  MoveL 3100 to (-5.96, 26.09, 135) mm, rotated rx -180 ry 0 rz 180 deg; joints [-155.969, -46.941, -94.947, 29.54, 55.687, -17.716]
  Call Extruder(28979.31277)
  MoveL 3101 to (-11.61, 24.12, 135) mm, rotated rx 180 ry 0 rz 180 deg; joints [-155.891, -46.52, -95.999, 29.42, 56.261, -17.391]
  Call Extruder(28988.67769)
  MoveL 3102 to (-16.69, 20.93, 135) mm, rotated rx 180 ry 0 rz -180 deg; joints [-156.025, -46.109, -97.037, 29.064, 56.768, -16.939]
  Call Extruder(28998.04290)
  MoveL 3103 to (-20.93, 16.69, 135) mm, rotated rx 180 ry 0 rz 180 deg; joints [-156.374, -45.729, -98.007, 28.481, 57.186, -16.384]
  Call Extruder(29007.40781)
  MoveL 3104 to (-24.11, 11.61, 135) mm, rotated rx 180 ry 0 rz 180 deg; joints [-156.928, -45.398, -98.859, 27.691, 57.492, -15.75]
  Call Extruder(29016.77261)
  MoveL 3105 to (-26.09, 5.96, 135) mm, rotated rx 180 ry 0 rz 180 deg; joints [-157.665, -45.134, -99.548, 26.726, 57.673, -15.07]
  Call Extruder(29026.13772)
  MoveL 3106 to (-26.77, 0, 135) mm, rotated rx -180 ry 0 rz 180 deg; joints [-158.546, -44.948, -100.034, 25.634, 57.719, -14.374]
  Call Extruder(29030.92646)
  MoveL 3107 to (-26.42, -3.05, 135) mm, rotated rx 180 ry 0 rz 180 deg; joints [-159.044, -44.897, -100.167, 25.04, 57.671, -14.027]
  Set speed (130.0 mm/s)
  MoveL 3108 to (-41.86, -6.29, 135) mm, rotated rx 180 ry 0 rz 180 deg; joints [-158.606, -43.913, -102.799, 25.112, 59.268, -13.469]
  Call Extruder(29035.92430)
  Set speed (60.0 mm/s)
  MoveL 3109 to (-41.51, -9.47, 135) mm, rotated rx 180 ry 0 rz 180 deg; joints [-159.151, -43.863, -102.935, 24.472, 59.22, -13.111]
  Call Extruder(29050.81995)
  MoveL 3110 to (-38.36, -18.47, 135) mm, rotated rx -180 ry 0 rz 180 deg; joints [-160.835, -43.856, -102.955, 22.553, 58.864, -12.119]
  Call Extruder(29065.71580)
  MoveL 3111 to (-33.28, -26.54, 135) mm, rotated rx 180 ry 0 rz 180 deg; joints [-162.466, -43.996, -102.574, 20.736, 58.31, -11.248]
  Call Extruder(29080.61162)
  MoveL 3112 to (-26.54, -33.28, 135) mm, rotated rx -180 ry 0 rz -180 deg; joints [-163.93, -44.276, -101.816, 19.142, 57.585, -10.54]
  Call Extruder(29095.50747)
  MoveL 3113 to (-18.47, -38.36, 135) mm, rotated rx 180 ry 0 rz 180 deg; joints [-165.137, -44.684, -100.729, 17.868, 56.725, -10.03]
  Call Extruder(29110.40312)
  MoveL 3114 to (-9.47, -41.51, 135) mm, rotated rx 180 ry 0 rz 180 deg; joints [-166.024, -45.2, -99.375, 16.984, 55.773, -9.748]
  Call Extruder(29125.29900)
  MoveL 3115 to (0, -42.57, 135) mm, rotated rx 180 ry 0 rz 180 deg; joints [-166.562, -45.797, -97.832, 16.528, 54.777, -9.712]
  Call Extruder(29140.19486)
  MoveL 3116 to (9.47, -41.51, 135) mm, rotated rx -180 ry 0 rz 180 deg; joints [-166.745, -46.447, -96.183, 16.51, 53.787, -9.932]
  Call Extruder(29155.09053)
  MoveL 3117 to (18.47, -38.36, 135) mm, rotated rx -180 ry 0 rz 180 deg; joints [-166.591, -47.117, -94.511, 16.913, 52.854, -10.405]
  Call Extruder(29169.98637)
  MoveL 3118 to (26.54, -33.28, 135) mm, rotated rx -180 ry 0 rz 180 deg; joints [-166.133, -47.772, -92.898, 17.701, 52.025, -11.111]
  Call Extruder(29184.88220)
  MoveL 3119 to (33.29, -26.54, 135) mm, rotated rx 180 ry 0 rz 180 deg; joints [-165.409, -48.38, -91.419, 18.819, 51.344, -12.018]
  Call Extruder(29199.77805)
  MoveL 3120 to (38.36, -18.47, 135) mm, rotated rx 180 ry 0 rz 180 deg; joints [-164.468, -48.911, -90.143, 20.202, 50.846, -13.08]
  Call Extruder(29214.67370)
  MoveL 3121 to (41.51, -9.47, 135) mm, rotated rx 180 ry 0 rz 180 deg; joints [-163.355, -49.337, -89.128, 21.772, 50.558, -14.238]
  Call Extruder(29229.56957)
  MoveL 3122 to (42.57, 0, 135) mm, rotated rx 180 ry 0 rz 180 deg; joints [-162.12, -49.636, -88.419, 23.448, 50.495, -15.425]
  Call Extruder(29244.46545)
  MoveL 3123 to (41.5, 9.47, 135) mm, rotated rx -180 ry 0 rz -180 deg; joints [-160.81, -49.793, -88.047, 25.15, 50.661, -16.574]
  Call Extruder(29259.36111)
  MoveL 3124 to (38.36, 18.47, 135) mm, rotated rx 180 ry 0 rz 180 deg; joints [-159.475, -49.801, -88.029, 26.8, 51.045, -17.619]
  Call Extruder(29274.25695)
  MoveL 3125 to (33.29, 26.54, 135) mm, rotated rx -180 ry 0 rz 180 deg; joints [-158.16, -49.658, -88.366, 28.328, 51.624, -18.504]
  Call Extruder(29289.15278)
  MoveL 3126 to (26.54, 33.28, 135) mm, rotated rx -180 ry 0 rz 180 deg; joints [-156.916, -49.372, -89.043, 29.675, 52.369, -19.184]
  Call Extruder(29304.04862)
  MoveL 3127 to (18.47, 38.36, 135) mm, rotated rx 180 ry 0 rz -180 deg; joints [-155.789, -48.958, -90.03, 30.791, 53.238, -19.628]
  Call Extruder(29318.94428)
  MoveL 3128 to (9.47, 41.51, 135) mm, rotated rx 180 ry 0 rz -180 deg; joints [-154.828, -48.437, -91.283, 31.635, 54.188, -19.822]
  Call Extruder(29333.84015)
  MoveL 3129 to (0, 42.57, 135) mm, rotated rx -180 ry 0 rz 180 deg; joints [-154.081, -47.835, -92.744, 32.174, 55.17, -19.764]
  Call Extruder(29348.73603)
  MoveL 3130 to (-9.47, 41.51, 135) mm, rotated rx 180 ry 0 rz -180 deg; joints [-153.594, -47.183, -94.347, 32.383, 56.137, -19.462]
  Call Extruder(29363.63168)
  MoveL 3131 to (-18.47, 38.36, 135) mm, rotated rx 180 ry 0 rz 180 deg; joints [-153.408, -46.513, -96.017, 32.24, 57.044, -18.937]
  Call Extruder(29378.52753)
  MoveL 3132 to (-26.54, 33.28, 135) mm, rotated rx -180 ry 0 rz 180 deg; joints [-153.557, -45.86, -97.672, 31.734, 57.847, -18.217]
  Call Extruder(29393.42335)
  MoveL 3133 to (-33.29, 26.54, 135) mm, rotated rx 180 ry 0 rz 180 deg; joints [-154.059, -45.256, -99.229, 30.864, 58.508, -17.338]
  Call Extruder(29408.31920)
  MoveL 3134 to (-38.36, 18.47, 135) mm, rotated rx 180 ry 0 rz 180 deg; joints [-154.913, -44.731, -100.605, 29.648, 58.995, -16.341]
  Call Extruder(29423.21486)
  MoveL 3135 to (-41.5, 9.47, 135) mm, rotated rx 180 ry 0 rz 180 deg; joints [-156.091, -44.311, -101.722, 28.127, 59.285, -15.271]
  Call Extruder(29438.11073)
  MoveL 3136 to (-42.57, 0, 135) mm, rotated rx 180 ry 0 rz -180 deg; joints [-157.533, -44.017, -102.515, 26.369, 59.362, -14.178]
  Call Extruder(29445.66501)
  MoveL 3137 to (-42.03, -4.8, 135) mm, rotated rx 180 ry 0 rz 180 deg; joints [-158.35, -43.937, -102.734, 25.411, 59.29, -13.637]
  Set speed (130.0 mm/s)
  MoveL 3138 to (-54.1, -7.67, 135) mm, rotated rx 180 ry 0 rz -180 deg; joints [-158.024, -43.197, -104.777, 25.454, 60.542, -13.175]
  Call Extruder(29449.73764)
  Set speed (30.0 mm/s)
  MoveL 3139 to (-53.59, -12.23, 135) mm, rotated rx 180 ry 0 rz 180 deg; joints [-158.835, -43.126, -104.975, 24.515, 60.477, -12.666]
  Call Extruder(29460.66777)
  MoveL 3140 to (-49.53, -23.85, 135) mm, rotated rx -180 ry 0 rz 180 deg; joints [-161.095, -43.117, -105.001, 21.965, 60.021, -11.394]
  Call Extruder(29471.59806)
  MoveL 3141 to (-42.98, -34.27, 135) mm, rotated rx 180 ry 0 rz 180 deg; joints [-163.275, -43.296, -104.498, 19.552, 59.308, -10.274]
  Call Extruder(29482.52818)
  MoveL 3142 to (-34.27, -42.98, 135) mm, rotated rx 180 ry 0 rz 180 deg; joints [-165.21, -43.657, -103.498, 17.446, 58.372, -9.358]
  Call Extruder(29493.45846)
  MoveL 3143 to (-23.85, -49.53, 135) mm, rotated rx -180 ry 0 rz -180 deg; joints [-166.774, -44.182, -102.069, 15.784, 57.261, -8.691]
  Call Extruder(29504.38859)
  MoveL 3144 to (-12.23, -53.59, 135) mm, rotated rx 180 ry 0 rz 180 deg; joints [-167.889, -44.847, -100.301, 14.654, 56.031, -8.313]
  Call Extruder(29515.31882)
  MoveL 3145 to (0, -54.97, 135) mm, rotated rx -180 ry 0 rz 180 deg; joints [-168.526, -45.617, -98.295, 14.099, 54.742, -8.25]
  Call Extruder(29524.69867)
  MoveL 3146 to (10.5, -53.79, 135) mm, rotated rx -180 ry 0 rz 180 deg; joints [-168.673, -46.335, -96.466, 14.115, 53.643, -8.479]
  Call Extruder(29526.24904)
  MoveL 3147 to (12.23, -53.59, 135) mm, rotated rx 180 ry 0 rz 180 deg; joints [-168.697, -46.456, -96.161, 14.12, 53.461, -8.517]
  Call Extruder(29537.17918)
  MoveL 3148 to (23.85, -49.53, 135) mm, rotated rx 180 ry 0 rz 180 deg; joints [-168.436, -47.32, -94.007, 14.685, 52.252, -9.115]
  Call Extruder(29548.10946)
  MoveL 3149 to (34.27, -42.98, 135) mm, rotated rx -180 ry 0 rz 180 deg; joints [-167.797, -48.167, -91.935, 15.743, 51.176, -10.022]
  Call Extruder(29559.03958)
  MoveL 3150 to (42.98, -34.27, 135) mm, rotated rx -180 ry 0 rz 180 deg; joints [-166.837, -48.954, -90.041, 17.218, 50.291, -11.199]
  Call Extruder(29569.96986)
  MoveL 3151 to (49.52, -23.85, 135) mm, rotated rx 180 ry 0 rz 180 deg; joints [-165.618, -49.64, -88.409, 19.023, 49.643, -12.585]
  Call Extruder(29580.89999)
  MoveL 3152 to (53.59, -12.23, 135) mm, rotated rx 180 ry 0 rz -180 deg; joints [-164.2, -50.191, -87.112, 21.058, 49.269, -14.103]
  Call Extruder(29591.83022)
  MoveL 3153 to (54.97, 0, 135) mm, rotated rx 180 ry 0 rz 180 deg; joints [-162.641, -50.579, -86.206, 23.217, 49.189, -15.66]
  Call Extruder(29602.76044)
  MoveL 3154 to (53.59, 12.23, 135) mm, rotated rx 180 ry 0 rz 180 deg; joints [-160.996, -50.782, -85.731, 25.393, 49.407, -17.164]
  Call Extruder(29613.69058)
  MoveL 3155 to (49.52, 23.85, 135) mm, rotated rx -180 ry 0 rz -180 deg; joints [-159.322, -50.792, -85.708, 27.489, 49.909, -18.525]
  Call Extruder(29624.62086)
  MoveL 3156 to (42.98, 34.27, 135) mm, rotated rx 180 ry 0 rz 180 deg; joints [-157.673, -50.607, -86.139, 29.418, 50.664, -19.668]
  Call Extruder(29635.55098)
  MoveL 3157 to (34.27, 42.98, 135) mm, rotated rx 180 ry 0 rz 180 deg; joints [-156.102, -50.237, -87.003, 31.111, 51.631, -20.536]
  Call Extruder(29646.48126)
  MoveL 3158 to (23.85, 49.53, 135) mm, rotated rx 180 ry 0 rz -180 deg; joints [-154.667, -49.701, -88.264, 32.512, 52.757, -21.093]
  Call Extruder(29657.41140)
  MoveL 3159 to (12.23, 53.59, 135) mm, rotated rx 180 ry 0 rz 180 deg; joints [-153.426, -49.027, -89.866, 33.578, 53.984, -21.323]
  Call Extruder(29668.34162)
  MoveL 3160 to (0, 54.97, 135) mm, rotated rx 180 ry 0 rz -180 deg; joints [-152.438, -48.249, -91.738, 34.274, 55.25, -21.229]
  Call Extruder(29679.27184)
  MoveL 3161 to (-12.23, 53.59, 135) mm, rotated rx 180 ry 0 rz -180 deg; joints [-151.764, -47.406, -93.796, 34.568, 56.494, -20.825]
  Call Extruder(29690.20198)
  MoveL 3162 to (-23.85, 49.52, 135) mm, rotated rx 180 ry 0 rz 180 deg; joints [-151.463, -46.541, -95.946, 34.432, 57.659, -20.14]
  Call Extruder(29701.13226)
  MoveL 3163 to (-34.27, 42.98, 135) mm, rotated rx 180 ry 0 rz 180 deg; joints [-151.589, -45.698, -98.087, 33.841, 58.691, -19.209]
  Call Extruder(29712.06238)
  MoveL 3164 to (-42.98, 34.27, 135) mm, rotated rx -180 ry 0 rz -180 deg; joints [-152.179, -44.919, -100.11, 32.78, 59.542, -18.078]
  Call Extruder(29722.99266)
  MoveL 3165 to (-49.53, 23.85, 135) mm, rotated rx 180 ry 0 rz 180 deg; joints [-153.248, -44.243, -101.907, 31.257, 60.172, -16.8]
  Call Extruder(29733.92280)
  MoveL 3166 to (-53.59, 12.23, 135) mm, rotated rx 180 ry 0 rz -180 deg; joints [-154.769, -43.702, -103.374, 29.309, 60.55, -15.43]
  Call Extruder(29744.85302)
  MoveL 3167 to (-54.97, 0, 135) mm, rotated rx 180 ry 0 rz -180 deg; joints [-156.673, -43.324, -104.42, 27.019, 60.654, -14.031]
  Call Extruder(29750.37864)
  MoveL 3168 to (-54.27, -6.18, 135) mm, rotated rx -180 ry 0 rz -180 deg; joints [-157.76, -43.221, -104.71, 25.759, 60.564, -13.341]
  Set speed (130.0 mm/s)
  MoveL 3169 to (-49.9, -9.51, 135) mm, rotated rx 180 ry 0 rz 180 deg; joints [-158.616, -43.388, -104.242, 24.873, 60.097, -13.014]
  MoveL 3170 to (2.97, -12.99, 135) mm, rotated rx 180 ry 0 rz -180 deg; joints [-162.152, -46.543, -95.942, 22.094, 54.573, -13.241]
  Call Extruder(29755.04223)
  Set speed (80.0 mm/s)
  MoveL 3171 to (5.78, -12.01, 135) mm, rotated rx 180 ry 0 rz 180 deg; joints [-162.141, -46.753, -95.417, 22.193, 54.284, -13.396]
  Call Extruder(29759.70584)
  MoveL 3172 to (8.31, -10.42, 135) mm, rotated rx 180 ry 0 rz -180 deg; joints [-162.027, -46.958, -94.906, 22.413, 54.027, -13.619]
  Call Extruder(29764.37004)
  MoveL 3173 to (10.42, -8.31, 135) mm, rotated rx -180 ry 0 rz 180 deg; joints [-161.819, -47.147, -94.434, 22.742, 53.816, -13.9]
  Call Extruder(29769.03367)
  MoveL 3174 to (12.01, -5.78, 135) mm, rotated rx 180 ry 0 rz 180 deg; joints [-161.529, -47.313, -94.025, 23.161, 53.662, -14.224]
  Call Extruder(29773.69724)
  MoveL 3175 to (12.99, -2.97, 135) mm, rotated rx -180 ry 0 rz -180 deg; joints [-161.171, -47.446, -93.698, 23.648, 53.573, -14.575]
  Call Extruder(29778.36118)
  MoveL 3176 to (13.33, 0, 135) mm, rotated rx 180 ry 0 rz 180 deg; joints [-160.763, -47.539, -93.469, 24.179, 53.553, -14.935]
  Call Extruder(29783.02514)
  MoveL 3177 to (12.99, 2.97, 135) mm, rotated rx -180 ry 0 rz 180 deg; joints [-160.324, -47.588, -93.348, 24.728, 53.602, -15.284]
  Call Extruder(29787.68872)
  MoveL 3178 to (12.01, 5.78, 135) mm, rotated rx 180 ry 0 rz -180 deg; joints [-159.874, -47.59, -93.343, 25.268, 53.719, -15.605]
  Call Extruder(29792.35234)
  MoveL 3179 to (10.42, 8.31, 135) mm, rotated rx -180 ry 0 rz 180 deg; joints [-159.432, -47.546, -93.452, 25.773, 53.897, -15.882]
  Call Extruder(29797.01653)
  MoveL 3180 to (8.31, 10.42, 135) mm, rotated rx -180 ry 0 rz 180 deg; joints [-159.021, -47.457, -93.67, 26.221, 54.127, -16.099]
  Call Extruder(29801.68015)
  MoveL 3181 to (5.78, 12.01, 135) mm, rotated rx -180 ry 0 rz 180 deg; joints [-158.657, -47.328, -93.989, 26.591, 54.398, -16.247]
  Call Extruder(29806.34373)
  MoveL 3182 to (2.97, 12.99, 135) mm, rotated rx 180 ry 0 rz 180 deg; joints [-158.359, -47.165, -94.39, 26.865, 54.695, -16.318]
  Call Extruder(29811.00768)
  MoveL 3183 to (0, 13.33, 135) mm, rotated rx 180 ry 0 rz 180 deg; joints [-158.143, -46.977, -94.857, 27.031, 55.004, -16.31]
  Call Extruder(29815.67163)
  MoveL 3184 to (-2.97, 13, 135) mm, rotated rx 180 ry 0 rz 180 deg; joints [-158.019, -46.773, -95.365, 27.079, 55.309, -16.224]
  Call Extruder(29820.33520)
  MoveL 3185 to (-5.78, 12.01, 135) mm, rotated rx 180 ry 0 rz 180 deg; joints [-157.997, -46.564, -95.89, 27.006, 55.596, -16.065]
  Call Extruder(29824.99883)
  MoveL 3186 to (-8.31, 10.42, 135) mm, rotated rx -180 ry 0 rz 180 deg; joints [-158.08, -46.359, -96.405, 26.813, 55.85, -15.84]
  Call Extruder(29829.66302)
  MoveL 3187 to (-10.42, 8.31, 135) mm, rotated rx 180 ry 0 rz 180 deg; joints [-158.266, -46.17, -96.884, 26.509, 56.059, -15.562]
  Call Extruder(29834.32664)
  MoveL 3188 to (-12.01, 5.78, 135) mm, rotated rx 180 ry 0 rz 180 deg; joints [-158.549, -46.005, -97.303, 26.106, 56.212, -15.244]
  Call Extruder(29838.99022)
  MoveL 3189 to (-12.99, 2.97, 135) mm, rotated rx 180 ry 0 rz -180 deg; joints [-158.913, -45.872, -97.641, 25.623, 56.302, -14.901]
  Call Extruder(29843.65417)
  MoveL 3190 to (-13.33, 0, 135) mm, rotated rx -180 ry 0 rz 180 deg; joints [-159.341, -45.78, -97.878, 25.084, 56.323, -14.551]
  Call Extruder(29848.31813)
  MoveL 3191 to (-13, -2.97, 135) mm, rotated rx 180 ry 0 rz -180 deg; joints [-159.811, -45.731, -98.003, 24.516, 56.276, -14.209]
  Call Extruder(29852.98169)
  MoveL 3192 to (-12.01, -5.78, 135) mm, rotated rx -180 ry 0 rz 180 deg; joints [-160.294, -45.729, -98.009, 23.951, 56.162, -13.893]
  Call Extruder(29857.64531)
  MoveL 3193 to (-10.42, -8.31, 135) mm, rotated rx 180 ry 0 rz 180 deg; joints [-160.766, -45.773, -97.895, 23.417, 55.986, -13.618]
  Call Extruder(29862.30952)
  MoveL 3194 to (-8.31, -10.42, 135) mm, rotated rx 180 ry 0 rz 180 deg; joints [-161.2, -45.861, -97.669, 22.945, 55.758, -13.398]
  Call Extruder(29866.97314)
  MoveL 3195 to (-5.78, -12.01, 135) mm, rotated rx -180 ry 0 rz 180 deg; joints [-161.572, -45.99, -97.341, 22.559, 55.489, -13.244]
  Call Extruder(29871.63671)
  MoveL 3196 to (-2.97, -13, 135) mm, rotated rx 180 ry 0 rz 180 deg; joints [-161.863, -46.152, -96.929, 22.281, 55.191, -13.164]
  Call Extruder(29876.30066)
  MoveL 3197 to (0, -13.33, 135) mm, rotated rx 180 ry 0 rz -180 deg; joints [-162.059, -46.34, -96.454, 22.123, 54.881, -13.163]
  Call Extruder(29880.96461)
  MoveL 3198 to (2.97, -12.99, 135) mm, rotated rx 180 ry 0 rz -180 deg; joints [-162.152, -46.543, -95.942, 22.094, 54.573, -13.241]
  Set speed (130.0 mm/s)
  MoveL 3199 to (2.97, -12.99, 140) mm, rotated rx -180 ry 0 rz -180 deg; joints [-162.152, -45.794, -96.186, 22.231, 54.106, -13.475]
  MoveL 3200 to (-26.25, -4.54, 140) mm, rotated rx 180 ry 0 rz 180 deg; joints [-159.288, -44.087, -100.482, 24.893, 57.163, -14.124]
  Call Extruder(29883.19722)
  Set speed (60.0 mm/s)
  MoveL 3201 to (-26.09, -5.96, 140) mm, rotated rx 180 ry 0 rz 180 deg; joints [-159.522, -44.064, -100.542, 24.614, 57.139, -13.959]
  Call Extruder(29892.56201)
  MoveL 3202 to (-24.12, -11.61, 140) mm, rotated rx -180 ry 0 rz 180 deg; joints [-160.532, -44.059, -100.554, 23.442, 56.908, -13.319]
  Call Extruder(29901.92694)
  MoveL 3203 to (-20.93, -16.69, 140) mm, rotated rx 180 ry 0 rz 180 deg; joints [-161.513, -44.149, -100.321, 22.334, 56.555, -12.758]
  Call Extruder(29911.29214)
  MoveL 3204 to (-16.69, -20.93, 140) mm, rotated rx 180 ry 0 rz 180 deg; joints [-162.406, -44.331, -99.856, 21.357, 56.098, -12.304]
  Call Extruder(29920.65706)
  MoveL 3205 to (-11.61, -24.12, 140) mm, rotated rx 180 ry 0 rz 180 deg; joints [-163.159, -44.595, -99.185, 20.566, 55.559, -11.98]
  Call Extruder(29930.02185)
  MoveL 3206 to (-5.96, -26.09, 140) mm, rotated rx 180 ry 0 rz 180 deg; joints [-163.733, -44.927, -98.346, 20.005, 54.965, -11.805]
  Call Extruder(29939.38695)
  MoveL 3207 to (0, -26.77, 140) mm, rotated rx -180 ry 0 rz 180 deg; joints [-164.103, -45.311, -97.383, 19.7, 54.346, -11.789]
  Call Extruder(29948.75206)
  MoveL 3208 to (5.96, -26.09, 140) mm, rotated rx -180 ry 0 rz 180 deg; joints [-164.258, -45.728, -96.348, 19.664, 53.733, -11.936]
  Call Extruder(29958.11686)
  MoveL 3209 to (11.61, -24.11, 140) mm, rotated rx 180 ry 0 rz 180 deg; joints [-164.201, -46.158, -95.294, 19.89, 53.156, -12.241]
  Call Extruder(29967.48177)
  MoveL 3210 to (16.69, -20.93, 140) mm, rotated rx 180 ry 0 rz 180 deg; joints [-163.944, -46.577, -94.271, 20.362, 52.646, -12.69]
  Call Extruder(29976.84698)
  MoveL 3211 to (20.93, -16.69, 140) mm, rotated rx -180 ry 0 rz 180 deg; joints [-163.508, -46.966, -93.331, 21.047, 52.228, -13.263]
  Call Extruder(29986.21190)
  MoveL 3212 to (24.12, -11.61, 140) mm, rotated rx 180 ry 0 rz 180 deg; joints [-162.92, -47.305, -92.518, 21.908, 51.925, -13.929]
  Call Extruder(29995.57669)
  MoveL 3213 to (26.09, -5.96, 140) mm, rotated rx 180 ry 0 rz -180 deg; joints [-162.209, -47.576, -91.87, 22.896, 51.752, -14.652]
  Call Extruder(30004.94180)
  MoveL 3214 to (26.77, 0, 140) mm, rotated rx 180 ry 0 rz -180 deg; joints [-161.41, -47.767, -91.416, 23.961, 51.717, -15.394]
  Call Extruder(30014.30690)
  MoveL 3215 to (26.09, 5.96, 140) mm, rotated rx 180 ry 0 rz 180 deg; joints [-160.556, -47.867, -91.178, 25.053, 51.824, -16.114]
  Call Extruder(30023.67170)
  MoveL 3216 to (24.12, 11.61, 140) mm, rotated rx 180 ry 0 rz 180 deg; joints [-159.683, -47.872, -91.167, 26.119, 52.065, -16.774]
  Call Extruder(30033.03662)
  MoveL 3217 to (20.93, 16.69, 140) mm, rotated rx 180 ry 0 rz 180 deg; joints [-158.826, -47.781, -91.382, 27.112, 52.428, -17.338]
  Call Extruder(30042.40183)
  MoveL 3218 to (16.69, 20.93, 140) mm, rotated rx 180 ry 0 rz 180 deg; joints [-158.019, -47.599, -91.815, 27.99, 52.894, -17.778]
  Call Extruder(30051.76674)
  MoveL 3219 to (11.61, 24.12, 140) mm, rotated rx 180 ry 0 rz 180 deg; joints [-157.299, -47.335, -92.446, 28.716, 53.438, -18.074]
  Call Extruder(30061.13154)
  MoveL 3220 to (5.96, 26.09, 140) mm, rotated rx 180 ry 0 rz -180 deg; joints [-156.697, -47.002, -93.244, 29.26, 54.033, -18.214]
  Call Extruder(30070.49665)
  MoveL 3221 to (0, 26.77, 140) mm, rotated rx 180 ry 0 rz 180 deg; joints [-156.245, -46.617, -94.174, 29.597, 54.649, -18.193]
  Call Extruder(30079.86174)
  MoveL 3222 to (-5.96, 26.09, 140) mm, rotated rx 180 ry 0 rz 180 deg; joints [-155.969, -46.2, -95.19, 29.709, 55.255, -18.015]
  Call Extruder(30089.22654)
  MoveL 3223 to (-11.61, 24.12, 140) mm, rotated rx -180 ry 0 rz -180 deg; joints [-155.891, -45.771, -96.244, 29.587, 55.821, -17.691]
  Call Extruder(30098.59146)
  MoveL 3224 to (-16.69, 20.93, 140) mm, rotated rx -180 ry 0 rz -180 deg; joints [-156.025, -45.351, -97.283, 29.229, 56.321, -17.238]
  Call Extruder(30107.95667)
  MoveL 3225 to (-20.93, 16.69, 140) mm, rotated rx -180 ry 0 rz 180 deg; joints [-156.374, -44.963, -98.255, 28.642, 56.73, -16.679]
  Call Extruder(30117.32158)
  MoveL 3226 to (-24.11, 11.61, 140) mm, rotated rx -180 ry 0 rz 180 deg; joints [-156.928, -44.625, -99.109, 27.848, 57.028, -16.041]
  Call Extruder(30126.68638)
  MoveL 3227 to (-26.09, 5.96, 140) mm, rotated rx 180 ry 0 rz -180 deg; joints [-157.665, -44.354, -99.798, 26.879, 57.2, -15.353]
  Call Extruder(30136.05148)
  MoveL 3228 to (-26.77, 0, 140) mm, rotated rx 180 ry 0 rz 180 deg; joints [-158.546, -44.163, -100.285, 25.781, 57.238, -14.648]
  Call Extruder(30140.84023)
  MoveL 3229 to (-26.42, -3.05, 140) mm, rotated rx 180 ry 0 rz 180 deg; joints [-159.044, -44.112, -100.419, 25.185, 57.187, -14.296]
  Set speed (130.0 mm/s)
  MoveL 3230 to (-41.86, -6.29, 140) mm, rotated rx 180 ry 0 rz 180 deg; joints [-158.606, -43.101, -103.056, 25.253, 58.766, -13.745]
  Call Extruder(30145.83807)
  Set speed (60.0 mm/s)
  MoveL 3231 to (-41.5, -9.47, 140) mm, rotated rx 180 ry 0 rz 180 deg; joints [-159.151, -43.05, -103.192, 24.611, 58.715, -13.381]
  Call Extruder(30160.73371)
  MoveL 3232 to (-38.36, -18.47, 140) mm, rotated rx 180 ry 0 rz 180 deg; joints [-160.835, -43.043, -103.212, 22.683, 58.351, -12.37]
  Call Extruder(30175.62957)
  MoveL 3233 to (-33.28, -26.54, 140) mm, rotated rx 180 ry 0 rz 180 deg; joints [-162.466, -43.187, -102.83, 20.859, 57.793, -11.48]
  Call Extruder(30190.52539)
  MoveL 3234 to (-26.54, -33.28, 140) mm, rotated rx 180 ry 0 rz -180 deg; joints [-163.93, -43.475, -102.071, 19.257, 57.068, -10.754]
  Call Extruder(30205.42124)
  MoveL 3235 to (-18.47, -38.36, 140) mm, rotated rx 180 ry 0 rz 180 deg; joints [-165.137, -43.893, -100.981, 17.977, 56.212, -10.229]
  Call Extruder(30220.31689)
  MoveL 3236 to (-9.47, -41.51, 140) mm, rotated rx -180 ry 0 rz 180 deg; joints [-166.024, -44.422, -99.625, 17.09, 55.267, -9.936]
  Call Extruder(30235.21276)
  MoveL 3237 to (0, -42.57, 140) mm, rotated rx -180 ry 0 rz 180 deg; joints [-166.562, -45.033, -98.08, 16.633, 54.281, -9.893]
  Call Extruder(30250.10864)
  MoveL 3238 to (9.47, -41.51, 140) mm, rotated rx -180 ry 0 rz -180 deg; joints [-166.745, -45.696, -96.428, 16.617, 53.302, -10.112]
  Call Extruder(30265.00430)
  MoveL 3239 to (18.47, -38.36, 140) mm, rotated rx -180 ry 0 rz 180 deg; joints [-166.591, -46.379, -94.753, 17.024, 52.38, -10.586]
  Call Extruder(30279.90014)
  MoveL 3240 to (26.54, -33.28, 140) mm, rotated rx 180 ry 0 rz 180 deg; joints [-166.133, -47.046, -93.138, 17.818, 51.563, -11.299]
  Call Extruder(30294.79596)
  MoveL 3241 to (33.29, -26.54, 140) mm, rotated rx 180 ry 0 rz 180 deg; joints [-165.409, -47.665, -91.658, 18.944, 50.893, -12.216]
  Call Extruder(30309.69181)
  MoveL 3242 to (38.36, -18.47, 140) mm, rotated rx -180 ry 0 rz 180 deg; joints [-164.468, -48.205, -90.381, 20.335, 50.406, -13.29]
  Call Extruder(30324.58747)
  MoveL 3243 to (41.5, -9.47, 140) mm, rotated rx 180 ry 0 rz 180 deg; joints [-163.355, -48.637, -89.365, 21.915, 50.128, -14.461]
  Call Extruder(30339.48334)
  MoveL 3244 to (42.57, 0, 140) mm, rotated rx 180 ry 0 rz 180 deg; joints [-162.12, -48.941, -88.655, 23.601, 50.075, -15.663]
  Call Extruder(30354.37921)
  MoveL 3245 to (41.51, 9.47, 140) mm, rotated rx -180 ry 0 rz 180 deg; joints [-160.81, -49.101, -88.283, 25.311, 50.248, -16.827]
  Call Extruder(30369.27488)
  MoveL 3246 to (38.36, 18.47, 140) mm, rotated rx -180 ry 0 rz 180 deg; joints [-159.475, -49.108, -88.265, 26.969, 50.637, -17.886]
  Call Extruder(30384.17072)
  MoveL 3247 to (33.28, 26.54, 140) mm, rotated rx -180 ry 0 rz 180 deg; joints [-158.16, -48.963, -88.602, 28.503, 51.221, -18.783]
  Call Extruder(30399.06654)
  MoveL 3248 to (26.54, 33.28, 140) mm, rotated rx 180 ry 0 rz 180 deg; joints [-156.916, -48.673, -89.28, 29.853, 51.967, -19.474]
  Call Extruder(30413.96239)
  MoveL 3249 to (18.47, 38.36, 140) mm, rotated rx 180 ry 0 rz -180 deg; joints [-155.789, -48.253, -90.268, 30.971, 52.836, -19.929]
  Call Extruder(30428.85805)
  MoveL 3250 to (9.47, 41.51, 140) mm, rotated rx -180 ry 0 rz 180 deg; joints [-154.828, -47.723, -91.521, 31.816, 53.783, -20.131]
  Call Extruder(30443.75392)
  MoveL 3251 to (0, 42.57, 140) mm, rotated rx 180 ry 0 rz 180 deg; joints [-154.081, -47.11, -92.984, 32.355, 54.761, -20.08]
  Call Extruder(30458.64980)
  MoveL 3252 to (-9.47, 41.51, 140) mm, rotated rx 180 ry 0 rz 180 deg; joints [-153.594, -46.446, -94.589, 32.562, 55.721, -19.782]
  Call Extruder(30473.54545)
  MoveL 3253 to (-18.47, 38.36, 140) mm, rotated rx 180 ry 0 rz 180 deg; joints [-153.408, -45.764, -96.261, 32.417, 56.617, -19.26]
  Call Extruder(30488.44130)
  MoveL 3254 to (-26.54, 33.29, 140) mm, rotated rx -180 ry 0 rz 180 deg; joints [-153.557, -45.097, -97.919, 31.907, 57.408, -18.54]
  Call Extruder(30503.33712)
  MoveL 3255 to (-33.28, 26.54, 140) mm, rotated rx 180 ry 0 rz 180 deg; joints [-154.059, -44.479, -99.479, 31.032, 58.055, -17.657]
  Call Extruder(30518.23296)
  MoveL 3256 to (-38.36, 18.47, 140) mm, rotated rx 180 ry 0 rz 180 deg; joints [-154.913, -43.941, -100.857, 29.81, 58.529, -16.652]
  Call Extruder(30533.12863)
  MoveL 3257 to (-41.5, 9.47, 140) mm, rotated rx -180 ry 0 rz 180 deg; joints [-156.091, -43.511, -101.977, 28.281, 58.804, -15.572]
  Call Extruder(30548.02450)
  MoveL 3258 to (-42.57, 0, 140) mm, rotated rx 180 ry 0 rz -180 deg; joints [-157.533, -43.209, -102.771, 26.516, 58.868, -14.465]
  Call Extruder(30555.57878)
  MoveL 3259 to (-42.03, -4.8, 140) mm, rotated rx 180 ry 0 rz 180 deg; joints [-158.35, -43.126, -102.99, 25.554, 58.79, -13.915]
  Set speed (130.0 mm/s)
  MoveL 3260 to (-54.1, -7.67, 140) mm, rotated rx 180 ry 0 rz 180 deg; joints [-158.024, -42.364, -105.038, 25.594, 60.027, -13.458]
  Call Extruder(30559.65141)
  Set speed (30.0 mm/s)
  MoveL 3261 to (-53.59, -12.23, 140) mm, rotated rx -180 ry 0 rz 180 deg; joints [-158.835, -42.292, -105.236, 24.651, 59.956, -12.94]
  Call Extruder(30570.58154)
  MoveL 3262 to (-49.52, -23.85, 140) mm, rotated rx 180 ry 0 rz 180 deg; joints [-161.095, -42.282, -105.263, 22.09, 59.49, -11.643]
  Call Extruder(30581.51183)
  MoveL 3263 to (-42.98, -34.27, 140) mm, rotated rx 180 ry 0 rz -180 deg; joints [-163.275, -42.467, -104.758, 19.666, 58.773, -10.497]
  Call Extruder(30592.44195)
  MoveL 3264 to (-34.27, -42.98, 140) mm, rotated rx 180 ry 0 rz 180 deg; joints [-165.21, -42.839, -103.756, 17.551, 57.838, -9.556]
  Call Extruder(30603.37223)
  MoveL 3265 to (-23.85, -49.53, 140) mm, rotated rx -180 ry 0 rz 180 deg; joints [-166.774, -43.378, -102.324, 15.881, 56.733, -8.87]
  Call Extruder(30614.30236)
  MoveL 3266 to (-12.23, -53.59, 140) mm, rotated rx -180 ry 0 rz 180 deg; joints [-167.889, -44.06, -100.552, 14.747, 55.513, -8.477]
  Call Extruder(30625.23259)
  MoveL 3267 to (0, -54.97, 140) mm, rotated rx -180 ry 0 rz 180 deg; joints [-168.526, -44.848, -98.543, 14.19, 54.237, -8.406]
  Call Extruder(30634.98527)
  MoveL 3268 to (10.91, -53.74, 140) mm, rotated rx -180 ry 0 rz 180 deg; joints [-168.679, -45.611, -96.638, 14.209, 53.107, -8.643]
  Call Extruder(30636.16281)
  MoveL 3269 to (12.23, -53.59, 140) mm, rotated rx -180 ry 0 rz 180 deg; joints [-168.697, -45.705, -96.406, 14.212, 52.971, -8.672]
  Call Extruder(30647.09295)
  MoveL 3270 to (23.85, -49.53, 140) mm, rotated rx 180 ry 0 rz 180 deg; joints [-168.436, -46.587, -94.249, 14.783, 51.776, -9.274]
  Call Extruder(30658.02323)
  MoveL 3271 to (34.27, -42.98, 140) mm, rotated rx -180 ry 0 rz 180 deg; joints [-167.797, -47.449, -92.174, 15.848, 50.715, -10.19]
  Call Extruder(30668.95335)
  MoveL 3272 to (42.98, -34.27, 140) mm, rotated rx 180 ry 0 rz 180 deg; joints [-166.837, -48.248, -90.278, 17.334, 49.844, -11.38]
  Call Extruder(30679.88363)
  MoveL 3273 to (49.53, -23.85, 140) mm, rotated rx -180 ry 0 rz 180 deg; joints [-165.618, -48.945, -88.645, 19.151, 49.209, -12.783]
  Call Extruder(30690.81376)
  MoveL 3274 to (53.59, -12.23, 140) mm, rotated rx -180 ry 0 rz -180 deg; joints [-164.2, -49.504, -87.347, 21.199, 48.848, -14.318]
  Call Extruder(30701.74399)
  MoveL 3275 to (54.97, 0, 140) mm, rotated rx -180 ry 0 rz 180 deg; joints [-162.641, -49.897, -86.44, 23.37, 48.779, -15.895]
  Call Extruder(30712.67421)
  MoveL 3276 to (53.59, 12.23, 140) mm, rotated rx -180 ry 0 rz 180 deg; joints [-160.996, -50.104, -85.965, 25.558, 49.006, -17.417]
  Call Extruder(30723.60435)
  MoveL 3277 to (49.52, 23.85, 140) mm, rotated rx 180 ry 0 rz -180 deg; joints [-159.322, -50.114, -85.942, 27.663, 49.515, -18.795]
  Call Extruder(30734.53463)
  MoveL 3278 to (42.98, 34.27, 140) mm, rotated rx 180 ry 0 rz 180 deg; joints [-157.673, -49.926, -86.373, 29.6, 50.276, -19.953]
  Call Extruder(30745.46475)
  MoveL 3279 to (34.27, 42.98, 140) mm, rotated rx -180 ry 0 rz 180 deg; joints [-156.102, -49.551, -87.238, 31.297, 51.245, -20.835]
  Call Extruder(30756.39503)
  MoveL 3280 to (23.85, 49.52, 140) mm, rotated rx 180 ry 0 rz 180 deg; joints [-154.667, -49.007, -88.5, 32.701, 52.371, -21.404]
  Call Extruder(30767.32517)
  MoveL 3281 to (12.23, 53.59, 140) mm, rotated rx 180 ry 0 rz 180 deg; joints [-153.426, -48.323, -90.103, 33.768, 53.595, -21.644]
  Call Extruder(30778.25539)
  MoveL 3282 to (0, 54.97, 140) mm, rotated rx 180 ry 0 rz 180 deg; joints [-152.438, -47.531, -91.977, 34.463, 54.855, -21.558]
  Call Extruder(30789.18561)
  MoveL 3283 to (-12.23, 53.59, 140) mm, rotated rx 180 ry 0 rz 180 deg; joints [-151.764, -46.674, -94.038, 34.754, 56.091, -21.16]
  Call Extruder(30800.11575)
  MoveL 3284 to (-23.85, 49.52, 140) mm, rotated rx 180 ry 0 rz 180 deg; joints [-151.463, -45.792, -96.191, 34.615, 57.243, -20.479]
  Call Extruder(30811.04603)
  MoveL 3285 to (-34.27, 42.98, 140) mm, rotated rx 180 ry 0 rz 180 deg; joints [-151.589, -44.931, -98.335, 34.019, 58.26, -19.549]
  Call Extruder(30821.97615)
  MoveL 3286 to (-42.98, 34.27, 140) mm, rotated rx 180 ry 0 rz -180 deg; joints [-152.179, -44.134, -100.362, 32.952, 59.093, -18.415]
  Call Extruder(30832.90643)
  MoveL 3287 to (-49.52, 23.85, 140) mm, rotated rx 180 ry 0 rz 180 deg; joints [-153.248, -43.44, -102.162, 31.422, 59.704, -17.129]
  Call Extruder(30843.83657)
  MoveL 3288 to (-53.59, 12.23, 140) mm, rotated rx -180 ry 0 rz 180 deg; joints [-154.769, -42.885, -103.632, 29.465, 60.062, -15.746]
  Call Extruder(30854.76679)
  MoveL 3289 to (-54.97, 0, 140) mm, rotated rx -180 ry 0 rz -180 deg; joints [-156.673, -42.496, -104.68, 27.165, 60.149, -14.329]
  Call Extruder(30860.29241)
  MoveL 3290 to (-54.27, -6.18, 140) mm, rotated rx 180 ry 0 rz 180 deg; joints [-157.76, -42.389, -104.971, 25.901, 60.051, -13.627]
  Set speed (130.0 mm/s)
  MoveL 3291 to (-49.9, -9.51, 140) mm, rotated rx 180 ry 0 rz 180 deg; joints [-158.616, -42.562, -104.502, 25.011, 59.584, -13.29]
  MoveL 3292 to (2.97, -12.99, 140) mm, rotated rx -180 ry 0 rz -180 deg; joints [-162.152, -45.794, -96.186, 22.231, 54.106, -13.475]
  Call Extruder(30864.95598)
  Set speed (80.0 mm/s)
  MoveL 3293 to (5.78, -12.01, 140) mm, rotated rx -180 ry 0 rz 180 deg; joints [-162.141, -46.008, -95.66, 22.331, 53.82, -13.63]
  Call Extruder(30869.61961)
  MoveL 3294 to (8.31, -10.42, 140) mm, rotated rx -180 ry 0 rz -180 deg; joints [-162.027, -46.217, -95.149, 22.553, 53.567, -13.855]
  Call Extruder(30874.28380)
  MoveL 3295 to (10.42, -8.31, 140) mm, rotated rx 180 ry 0 rz 180 deg; joints [-161.819, -46.41, -94.677, 22.883, 53.36, -14.138]
  Call Extruder(30878.94743)
  MoveL 3296 to (12.01, -5.78, 140) mm, rotated rx 180 ry 0 rz 180 deg; joints [-161.529, -46.579, -94.267, 23.305, 53.21, -14.466]
  Call Extruder(30883.61100)
  MoveL 3297 to (13, -2.97, 140) mm, rotated rx 180 ry 0 rz -180 deg; joints [-161.171, -46.714, -93.939, 23.795, 53.124, -14.821]
  Call Extruder(30888.27495)
  MoveL 3298 to (13.33, 0, 140) mm, rotated rx -180 ry 0 rz 180 deg; joints [-160.763, -46.809, -93.71, 24.329, 53.107, -15.185]
  Call Extruder(30892.93890)
  MoveL 3299 to (13, 2.97, 140) mm, rotated rx 180 ry 0 rz 180 deg; joints [-160.324, -46.859, -93.589, 24.88, 53.159, -15.539]
  Call Extruder(30897.60248)
  MoveL 3300 to (12.01, 5.78, 140) mm, rotated rx 180 ry 0 rz -180 deg; joints [-159.874, -46.861, -93.584, 25.422, 53.278, -15.865]
  Call Extruder(30902.26610)
  MoveL 3301 to (10.42, 8.31, 140) mm, rotated rx 180 ry 0 rz 180 deg; joints [-159.432, -46.816, -93.693, 25.93, 53.457, -16.146]
  Call Extruder(30906.93029)
  MoveL 3302 to (8.31, 10.42, 140) mm, rotated rx 180 ry 0 rz 180 deg; joints [-159.021, -46.726, -93.912, 26.38, 53.688, -16.367]
  Call Extruder(30911.59391)
  MoveL 3303 to (5.78, 12.01, 140) mm, rotated rx -180 ry 0 rz 180 deg; joints [-158.657, -46.594, -94.23, 26.75, 53.958, -16.519]
  Call Extruder(30916.25749)
  MoveL 3304 to (2.97, 13, 140) mm, rotated rx 180 ry 0 rz 180 deg; joints [-158.359, -46.428, -94.633, 27.025, 54.254, -16.593]
  Call Extruder(30920.92145)
  MoveL 3305 to (0, 13.33, 140) mm, rotated rx 180 ry 0 rz 180 deg; joints [-158.143, -46.237, -95.1, 27.191, 54.561, -16.588]
  Call Extruder(30925.58539)
  MoveL 3306 to (-2.97, 12.99, 140) mm, rotated rx -180 ry 0 rz 180 deg; joints [-158.019, -46.029, -95.609, 27.238, 54.864, -16.503]
  Call Extruder(30930.24896)
  MoveL 3307 to (-5.78, 12.01, 140) mm, rotated rx -180 ry 0 rz -180 deg; joints [-157.997, -45.815, -96.134, 27.164, 55.147, -16.344]
  Call Extruder(30934.91259)
  MoveL 3308 to (-8.31, 10.42, 140) mm, rotated rx 180 ry 0 rz 180 deg; joints [-158.08, -45.606, -96.65, 26.971, 55.398, -16.118]
  Call Extruder(30939.57679)
  MoveL 3309 to (-10.42, 8.31, 140) mm, rotated rx -180 ry 0 rz 180 deg; joints [-158.266, -45.413, -97.13, 26.664, 55.602, -15.838]
  Call Extruder(30944.24041)
  MoveL 3310 to (-12.01, 5.78, 140) mm, rotated rx -180 ry 0 rz 180 deg; joints [-158.549, -45.244, -97.55, 26.259, 55.751, -15.517]
  Call Extruder(30948.90398)
  MoveL 3311 to (-12.99, 2.97, 140) mm, rotated rx 180 ry 0 rz -180 deg; joints [-158.913, -45.109, -97.888, 25.774, 55.837, -15.171]
  Call Extruder(30953.56793)
  MoveL 3312 to (-13.33, 0, 140) mm, rotated rx 180 ry 0 rz 180 deg; joints [-159.341, -45.014, -98.125, 25.232, 55.855, -14.816]
  Call Extruder(30958.23189)
  MoveL 3313 to (-13, -2.97, 140) mm, rotated rx -180 ry 0 rz 180 deg; joints [-159.811, -44.965, -98.251, 24.662, 55.804, -14.469]
  Call Extruder(30962.89545)
  MoveL 3314 to (-12.01, -5.78, 140) mm, rotated rx 180 ry 0 rz 180 deg; joints [-160.294, -44.962, -98.256, 24.093, 55.688, -14.148]
  Call Extruder(30967.55908)
  MoveL 3315 to (-10.42, -8.31, 140) mm, rotated rx 180 ry 0 rz 180 deg; joints [-160.766, -45.007, -98.143, 23.557, 55.511, -13.868]
  Call Extruder(30972.22328)
  MoveL 3316 to (-8.31, -10.42, 140) mm, rotated rx 180 ry 0 rz 180 deg; joints [-161.2, -45.098, -97.916, 23.083, 55.283, -13.643]
  Call Extruder(30976.88691)
  MoveL 3317 to (-5.78, -12.01, 140) mm, rotated rx -180 ry 0 rz 180 deg; joints [-161.572, -45.229, -97.587, 22.696, 55.014, -13.485]
  Call Extruder(30981.55047)
  MoveL 3318 to (-2.97, -12.99, 140) mm, rotated rx -180 ry 0 rz 180 deg; joints [-161.863, -45.395, -97.175, 22.417, 54.718, -13.402]
  Call Extruder(30986.21442)
  MoveL 3319 to (0, -13.33, 140) mm, rotated rx -180 ry 0 rz -180 deg; joints [-162.059, -45.586, -96.7, 22.259, 54.41, -13.398]
  Call Extruder(30990.87838)
  MoveL 3320 to (2.97, -12.99, 140) mm, rotated rx -180 ry 0 rz -180 deg; joints [-162.152, -45.794, -96.186, 22.231, 54.106, -13.475]
  Set speed (130.0 mm/s)
  MoveL 3321 to (2.97, -12.99, 145) mm, rotated rx -180 ry 0 rz -180 deg; joints [-162.152, -45.047, -96.421, 22.372, 53.632, -13.716]
  MoveL 3322 to (-26.25, -4.54, 145) mm, rotated rx 180 ry 0 rz 180 deg; joints [-159.288, -43.302, -100.724, 25.042, 56.671, -14.397]
  Call Extruder(30993.11100)
  Set speed (60.0 mm/s)
  MoveL 3323 to (-26.09, -5.96, 145) mm, rotated rx 180 ry 0 rz 180 deg; joints [-159.522, -43.278, -100.784, 24.762, 56.646, -14.23]
  Call Extruder(31002.47579)
  MoveL 3324 to (-24.12, -11.61, 145) mm, rotated rx -180 ry 0 rz 180 deg; joints [-160.532, -43.273, -100.796, 23.584, 56.41, -13.579]
  Call Extruder(31011.84071)
  MoveL 3325 to (-20.93, -16.69, 145) mm, rotated rx -180 ry 0 rz 180 deg; joints [-161.513, -43.366, -100.563, 22.472, 56.054, -13.006]
  Call Extruder(31021.20591)
  MoveL 3326 to (-16.69, -20.93, 145) mm, rotated rx 180 ry 0 rz 180 deg; joints [-162.406, -43.552, -100.097, 21.49, 55.597, -12.541]
  Call Extruder(31030.57084)
  MoveL 3327 to (-11.61, -24.12, 145) mm, rotated rx 180 ry 0 rz 180 deg; joints [-163.159, -43.822, -99.424, 20.696, 55.06, -12.209]
  Call Extruder(31039.93563)
  MoveL 3328 to (-5.96, -26.09, 145) mm, rotated rx -180 ry 0 rz -180 deg; joints [-163.733, -44.162, -98.584, 20.133, 54.47, -12.026]
  Call Extruder(31049.30073)
  MoveL 3329 to (0, -26.77, 145) mm, rotated rx -180 ry 0 rz 180 deg; joints [-164.103, -44.554, -97.62, 19.827, 53.856, -12.006]
  Call Extruder(31058.66583)
  MoveL 3330 to (5.96, -26.09, 145) mm, rotated rx 180 ry 0 rz 180 deg; joints [-164.258, -44.98, -96.583, 19.792, 53.25, -12.151]
  Call Extruder(31068.03064)
  MoveL 3331 to (11.61, -24.11, 145) mm, rotated rx 180 ry 0 rz 180 deg; joints [-164.201, -45.418, -95.527, 20.021, 52.68, -12.457]
  Call Extruder(31077.39555)
  MoveL 3332 to (16.69, -20.93, 145) mm, rotated rx -180 ry 0 rz 180 deg; joints [-163.944, -45.845, -94.504, 20.496, 52.178, -12.91]
  Call Extruder(31086.76076)
  MoveL 3333 to (20.93, -16.69, 145) mm, rotated rx 180 ry 0 rz 180 deg; joints [-163.508, -46.241, -93.563, 21.186, 51.768, -13.489]
  Call Extruder(31096.12568)
  MoveL 3334 to (24.12, -11.61, 145) mm, rotated rx -180 ry 0 rz 180 deg; joints [-162.92, -46.586, -92.748, 22.052, 51.472, -14.162]
  Call Extruder(31105.49047)
  MoveL 3335 to (26.09, -5.96, 145) mm, rotated rx 180 ry 0 rz -180 deg; joints [-162.209, -46.862, -92.099, 23.046, 51.306, -14.894]
  Call Extruder(31114.85557)
  MoveL 3336 to (26.77, 0, 145) mm, rotated rx -180 ry 0 rz -180 deg; joints [-161.41, -47.056, -91.645, 24.118, 51.277, -15.645]
  Call Extruder(31124.22068)
  MoveL 3337 to (26.09, 5.96, 145) mm, rotated rx 180 ry 0 rz 180 deg; joints [-160.556, -47.158, -91.407, 25.214, 51.389, -16.375]
  Call Extruder(31133.58548)
  MoveL 3338 to (24.12, 11.61, 145) mm, rotated rx 180 ry 0 rz 180 deg; joints [-159.683, -47.163, -91.395, 26.285, 51.634, -17.043]
  Call Extruder(31142.95039)
  MoveL 3339 to (20.93, 16.69, 145) mm, rotated rx 180 ry 0 rz 180 deg; joints [-158.826, -47.071, -91.611, 27.283, 52, -17.616]
  Call Extruder(31152.31560)
  MoveL 3340 to (16.69, 20.93, 145) mm, rotated rx -180 ry 0 rz 180 deg; joints [-158.019, -46.886, -92.045, 28.164, 52.467, -18.065]
  Call Extruder(31161.68051)
  MoveL 3341 to (11.61, 24.12, 145) mm, rotated rx 180 ry 0 rz 180 deg; joints [-157.299, -46.617, -92.676, 28.892, 53.011, -18.368]
  Call Extruder(31171.04532)
  MoveL 3342 to (5.96, 26.09, 145) mm, rotated rx 180 ry 0 rz 180 deg; joints [-156.697, -46.278, -93.475, 29.437, 53.603, -18.513]
  Call Extruder(31180.41042)
  MoveL 3343 to (0, 26.77, 145) mm, rotated rx 180 ry 0 rz 180 deg; joints [-156.245, -45.886, -94.406, 29.774, 54.215, -18.497]
  Call Extruder(31189.77552)
  MoveL 3344 to (-5.96, 26.09, 145) mm, rotated rx 180 ry 0 rz 180 deg; joints [-155.969, -45.461, -95.423, 29.885, 54.816, -18.321]
  Call Extruder(31199.14031)
  MoveL 3345 to (-11.61, 24.12, 145) mm, rotated rx 180 ry 0 rz 180 deg; joints [-155.891, -45.023, -96.479, 29.761, 55.376, -17.998]
  Call Extruder(31208.50523)
  MoveL 3346 to (-16.69, 20.93, 145) mm, rotated rx 180 ry 0 rz -180 deg; joints [-156.025, -44.595, -97.519, 29.4, 55.868, -17.545]
  Call Extruder(31217.87044)
  MoveL 3347 to (-20.93, 16.69, 145) mm, rotated rx 180 ry 0 rz 180 deg; joints [-156.374, -44.198, -98.493, 28.81, 56.268, -16.983]
  Call Extruder(31227.23535)
  MoveL 3348 to (-24.11, 11.61, 145) mm, rotated rx -180 ry 0 rz 180 deg; joints [-156.928, -43.853, -99.348, 28.011, 56.557, -16.339]
  Call Extruder(31236.60015)
  MoveL 3349 to (-26.09, 5.96, 145) mm, rotated rx 180 ry 0 rz 180 deg; joints [-157.665, -43.575, -100.038, 27.037, 56.721, -15.644]
  Call Extruder(31245.96526)
  MoveL 3350 to (-26.77, 0, 145) mm, rotated rx 180 ry 0 rz 180 deg; joints [-158.546, -43.381, -100.526, 25.935, 56.751, -14.93]
  Call Extruder(31250.75400)
  MoveL 3351 to (-26.42, -3.05, 145) mm, rotated rx 180 ry 0 rz 180 deg; joints [-159.044, -43.327, -100.66, 25.336, 56.697, -14.572]
  Set speed (130.0 mm/s)
  MoveL 3352 to (-41.86, -6.29, 145) mm, rotated rx 180 ry 0 rz 180 deg; joints [-158.606, -42.291, -103.303, 25.401, 58.257, -14.027]
  Call Extruder(31255.75184)
  Set speed (60.0 mm/s)
  MoveL 3353 to (-41.5, -9.47, 145) mm, rotated rx -180 ry 0 rz 180 deg; joints [-159.151, -42.239, -103.439, 24.756, 58.202, -13.657]
  Call Extruder(31270.64749)
  MoveL 3354 to (-38.36, -18.47, 145) mm, rotated rx -180 ry 0 rz -180 deg; joints [-160.835, -42.231, -103.459, 22.819, 57.83, -12.627]
  Call Extruder(31285.54334)
  MoveL 3355 to (-33.28, -26.54, 145) mm, rotated rx 180 ry 0 rz 180 deg; joints [-162.466, -42.379, -103.077, 20.986, 57.269, -11.717]
  Call Extruder(31300.43916)
  MoveL 3356 to (-26.54, -33.28, 145) mm, rotated rx 180 ry 0 rz -180 deg; joints [-163.93, -42.675, -102.316, 19.377, 56.544, -10.973]
  Call Extruder(31315.33501)
  MoveL 3357 to (-18.47, -38.36, 145) mm, rotated rx 180 ry 0 rz 180 deg; joints [-165.137, -43.104, -101.224, 18.092, 55.692, -10.433]
  Call Extruder(31330.23066)
  MoveL 3358 to (-9.47, -41.5, 145) mm, rotated rx -180 ry 0 rz 180 deg; joints [-166.024, -43.645, -99.865, 17.201, 54.755, -10.129]
  Call Extruder(31345.12654)
  MoveL 3359 to (0, -42.57, 145) mm, rotated rx -180 ry 0 rz 180 deg; joints [-166.562, -44.27, -98.317, 16.742, 53.778, -10.08]
  Call Extruder(31360.02241)
  MoveL 3360 to (9.47, -41.51, 145) mm, rotated rx -180 ry 0 rz 180 deg; joints [-166.745, -44.947, -96.663, 16.727, 52.81, -10.296]
  Call Extruder(31374.91807)
  MoveL 3361 to (18.47, -38.36, 145) mm, rotated rx -180 ry 0 rz 180 deg; joints [-166.591, -45.643, -94.986, 17.138, 51.9, -10.773]
  Call Extruder(31389.81392)
  MoveL 3362 to (26.54, -33.28, 145) mm, rotated rx 180 ry 0 rz 180 deg; joints [-166.133, -46.323, -93.369, 17.938, 51.094, -11.493]
  Call Extruder(31404.70974)
  MoveL 3363 to (33.29, -26.54, 145) mm, rotated rx 180 ry 0 rz 180 deg; joints [-165.409, -46.953, -91.887, 19.073, 50.436, -12.419]
  Call Extruder(31419.60559)
  MoveL 3364 to (38.36, -18.47, 145) mm, rotated rx 180 ry 0 rz 180 deg; joints [-164.468, -47.501, -90.609, 20.473, 49.96, -13.506]
  Call Extruder(31434.50124)
  MoveL 3365 to (41.51, -9.47, 145) mm, rotated rx -180 ry 0 rz 180 deg; joints [-163.355, -47.94, -89.592, 22.063, 49.693, -14.691]
  Call Extruder(31449.39711)
  MoveL 3366 to (42.57, 0, 145) mm, rotated rx 180 ry 0 rz 180 deg; joints [-162.12, -48.248, -88.881, 23.758, 49.648, -15.908]
  Call Extruder(31464.29299)
  MoveL 3367 to (41.51, 9.47, 145) mm, rotated rx 180 ry 0 rz 180 deg; joints [-160.81, -48.411, -88.509, 25.478, 49.829, -17.086]
  Call Extruder(31479.18865)
  MoveL 3368 to (38.36, 18.47, 145) mm, rotated rx -180 ry 0 rz 180 deg; joints [-159.475, -48.418, -88.491, 27.143, 50.224, -18.159]
  Call Extruder(31494.08449)
  MoveL 3369 to (33.29, 26.54, 145) mm, rotated rx 180 ry 0 rz 180 deg; joints [-158.16, -48.271, -88.829, 28.683, 50.812, -19.07]
  Call Extruder(31508.98032)
  MoveL 3370 to (26.54, 33.29, 145) mm, rotated rx 180 ry 0 rz -180 deg; joints [-156.916, -47.977, -89.507, 30.038, 51.561, -19.773]
  Call Extruder(31523.87616)
  MoveL 3371 to (18.47, 38.36, 145) mm, rotated rx -180 ry 0 rz -180 deg; joints [-155.789, -47.55, -90.496, 31.159, 52.429, -20.237]
  Call Extruder(31538.77182)
  MoveL 3372 to (9.47, 41.51, 145) mm, rotated rx 180 ry 0 rz 180 deg; joints [-154.828, -47.011, -91.751, 32.004, 53.374, -20.448]
  Call Extruder(31553.66770)
  MoveL 3373 to (0, 42.57, 145) mm, rotated rx 180 ry 0 rz 180 deg; joints [-154.081, -46.388, -93.215, 32.543, 54.346, -20.403]
  Call Extruder(31568.56357)
  MoveL 3374 to (-9.47, 41.51, 145) mm, rotated rx 180 ry 0 rz 180 deg; joints [-153.594, -45.712, -94.822, 32.748, 55.298, -20.111]
  Call Extruder(31583.45922)
  MoveL 3375 to (-18.47, 38.36, 145) mm, rotated rx 180 ry 0 rz 180 deg; joints [-153.408, -45.016, -96.496, 32.6, 56.185, -19.591]
  Call Extruder(31598.35507)
  MoveL 3376 to (-26.54, 33.29, 145) mm, rotated rx 180 ry 0 rz 180 deg; joints [-153.557, -44.335, -98.157, 32.086, 56.963, -18.87]
  Call Extruder(31613.25089)
  MoveL 3377 to (-33.28, 26.54, 145) mm, rotated rx -180 ry 0 rz 180 deg; joints [-154.059, -43.704, -99.719, 31.206, 57.597, -17.984]
  Call Extruder(31628.14674)
  MoveL 3378 to (-38.36, 18.47, 145) mm, rotated rx 180 ry 0 rz 180 deg; joints [-154.913, -43.153, -101.1, 29.978, 58.055, -16.972]
  Call Extruder(31643.04240)
  MoveL 3379 to (-41.5, 9.47, 145) mm, rotated rx -180 ry 0 rz 180 deg; joints [-156.091, -42.712, -102.221, 28.442, 58.316, -15.881]
  Call Extruder(31657.93828)
  MoveL 3380 to (-42.57, 0, 145) mm, rotated rx -180 ry 0 rz -180 deg; joints [-157.533, -42.402, -103.017, 26.67, 58.366, -14.759]
  Call Extruder(31665.49256)
  MoveL 3381 to (-42.03, -4.8, 145) mm, rotated rx 180 ry 0 rz 180 deg; joints [-158.35, -42.317, -103.237, 25.703, 58.282, -14.201]
  Set speed (130.0 mm/s)
  MoveL 3382 to (-54.1, -7.67, 145) mm, rotated rx 180 ry 0 rz 180 deg; joints [-158.024, -41.533, -105.289, 25.741, 59.504, -13.749]
  Call Extruder(31669.56519)
  Set speed (30.0 mm/s)
  MoveL 3383 to (-53.59, -12.23, 145) mm, rotated rx 180 ry 0 rz 180 deg; joints [-158.835, -41.459, -105.488, 24.794, 59.427, -13.222]
  Call Extruder(31680.49532)
  MoveL 3384 to (-49.53, -23.85, 145) mm, rotated rx 180 ry 0 rz 180 deg; joints [-161.095, -41.449, -105.515, 22.221, 58.951, -11.898]
  Call Extruder(31691.42560)
  MoveL 3385 to (-42.98, -34.27, 145) mm, rotated rx 180 ry 0 rz -180 deg; joints [-163.275, -41.639, -105.008, 19.786, 58.229, -10.725]
  Call Extruder(31702.35572)
  MoveL 3386 to (-34.27, -42.98, 145) mm, rotated rx 180 ry 0 rz -180 deg; joints [-165.21, -42.022, -104.004, 17.66, 57.296, -9.76]
  Call Extruder(31713.28600)
  MoveL 3387 to (-23.85, -49.52, 145) mm, rotated rx 180 ry 0 rz 180 deg; joints [-166.774, -42.576, -102.57, 15.982, 56.197, -9.053]
  Call Extruder(31724.21614)
  MoveL 3388 to (-12.23, -53.59, 145) mm, rotated rx 180 ry 0 rz -180 deg; joints [-167.889, -43.274, -100.794, 14.843, 54.987, -8.646]
  Call Extruder(31735.14636)
  MoveL 3389 to (0, -54.97, 145) mm, rotated rx 180 ry 0 rz 180 deg; joints [-168.526, -44.081, -98.782, 14.285, 53.725, -8.567]
  Call Extruder(31741.60007)
  MoveL 3390 to (7.22, -54.16, 145) mm, rotated rx 180 ry 0 rz 180 deg; joints [-168.628, -44.594, -97.522, 14.296, 52.986, -8.721]
  Call Extruder(31746.07658)
  MoveL 3391 to (12.23, -53.59, 145) mm, rotated rx 180 ry 0 rz 180 deg; joints [-168.697, -44.956, -96.641, 14.309, 52.473, -8.831]
  Call Extruder(31757.00672)
  MoveL 3392 to (23.85, -49.53, 145) mm, rotated rx -180 ry 0 rz 180 deg; joints [-168.436, -45.855, -94.481, 14.885, 51.293, -9.437]
  Call Extruder(31767.93700)
  MoveL 3393 to (34.27, -42.98, 145) mm, rotated rx 180 ry 0 rz 180 deg; joints [-167.797, -46.732, -92.404, 15.958, 50.247, -10.363]
  Call Extruder(31778.86712)
  MoveL 3394 to (42.98, -34.27, 145) mm, rotated rx -180 ry 0 rz 180 deg; joints [-166.837, -47.545, -90.506, 17.455, 49.39, -11.567]
  Call Extruder(31789.79740)
  MoveL 3395 to (49.52, -23.85, 145) mm, rotated rx -180 ry 0 rz 180 deg; joints [-165.618, -48.253, -88.872, 19.285, 48.77, -12.986]
  Call Extruder(31800.72754)
  MoveL 3396 to (53.59, -12.23, 145) mm, rotated rx 180 ry 0 rz -180 deg; joints [-164.2, -48.82, -87.572, 21.346, 48.42, -14.54]
  Call Extruder(31811.65776)
  MoveL 3397 to (54.97, 0, 145) mm, rotated rx 180 ry 0 rz 180 deg; joints [-162.641, -49.218, -86.665, 23.53, 48.363, -16.135]
  Call Extruder(31822.58798)
  MoveL 3398 to (53.59, 12.23, 145) mm, rotated rx -180 ry 0 rz 180 deg; joints [-160.996, -49.428, -86.19, 25.729, 48.599, -17.676]
  Call Extruder(31833.51813)
  MoveL 3399 to (49.52, 23.85, 145) mm, rotated rx -180 ry 0 rz -180 deg; joints [-159.322, -49.438, -86.167, 27.844, 49.116, -19.072]
  Call Extruder(31844.44840)
  MoveL 3400 to (42.98, 34.27, 145) mm, rotated rx 180 ry 0 rz 180 deg; joints [-157.673, -49.248, -86.598, 29.787, 49.882, -20.246]
  Call Extruder(31855.37853)
  MoveL 3401 to (34.27, 42.98, 145) mm, rotated rx -180 ry 0 rz 180 deg; joints [-156.102, -48.867, -87.464, 31.49, 50.855, -21.142]
  Call Extruder(31866.30880)
  MoveL 3402 to (23.85, 49.52, 145) mm, rotated rx 180 ry 0 rz -180 deg; joints [-154.667, -48.316, -88.727, 32.896, 51.981, -21.723]
  Call Extruder(31877.23894)
  MoveL 3403 to (12.23, 53.59, 145) mm, rotated rx 180 ry 0 rz 180 deg; joints [-153.426, -47.621, -90.331, 33.964, 53.202, -21.973]
  Call Extruder(31888.16917)
  MoveL 3404 to (0, 54.97, 145) mm, rotated rx 180 ry 0 rz -180 deg; joints [-152.438, -46.817, -92.207, 34.658, 54.456, -21.895]
  Call Extruder(31899.09939)
  MoveL 3405 to (-12.23, 53.59, 145) mm, rotated rx 180 ry 0 rz 180 deg; joints [-151.764, -45.944, -94.27, 34.947, 55.682, -21.504]
  Call Extruder(31910.02952)
  MoveL 3406 to (-23.85, 49.52, 145) mm, rotated rx 180 ry 0 rz 180 deg; joints [-151.463, -45.045, -96.426, 34.804, 56.822, -20.826]
  Call Extruder(31920.95980)
  MoveL 3407 to (-34.27, 42.98, 145) mm, rotated rx 180 ry 0 rz 180 deg; joints [-151.589, -44.166, -98.573, 34.203, 57.824, -19.897]
  Call Extruder(31931.88992)
  MoveL 3408 to (-42.98, 34.27, 145) mm, rotated rx 180 ry 0 rz -180 deg; joints [-152.179, -43.35, -100.603, 33.131, 58.639, -18.761]
  Call Extruder(31942.82020)
  MoveL 3409 to (-49.52, 23.85, 145) mm, rotated rx 180 ry 0 rz 180 deg; joints [-153.248, -42.639, -102.407, 31.593, 59.23, -17.466]
  Call Extruder(31953.75035)
  MoveL 3410 to (-53.59, 12.23, 145) mm, rotated rx 180 ry 0 rz -180 deg; joints [-154.769, -42.069, -103.88, 29.628, 59.568, -16.07]
  Call Extruder(31964.68057)
  MoveL 3411 to (-54.97, 0, 145) mm, rotated rx -180 ry 0 rz -180 deg; joints [-156.673, -41.669, -104.93, 27.319, 59.636, -14.634]
  Call Extruder(31970.20619)
  MoveL 3412 to (-54.27, -6.18, 145) mm, rotated rx 180 ry 0 rz 180 deg; joints [-157.76, -41.559, -105.222, 26.049, 59.53, -13.921]
  Set speed (130.0 mm/s)
  MoveL 3413 to (-49.9, -9.51, 145) mm, rotated rx 180 ry 0 rz -180 deg; joints [-158.616, -41.737, -104.752, 25.156, 59.063, -13.574]
  MoveL 3414 to (2.97, -12.99, 145) mm, rotated rx -180 ry 0 rz -180 deg; joints [-162.152, -45.047, -96.421, 22.372, 53.632, -13.716]
  Call Extruder(31974.86976)
  Set speed (80.0 mm/s)
  MoveL 3415 to (5.78, -12.01, 145) mm, rotated rx -180 ry 0 rz 180 deg; joints [-162.141, -45.265, -95.895, 22.474, 53.35, -13.871]
  Call Extruder(31979.53339)
  MoveL 3416 to (8.31, -10.42, 145) mm, rotated rx 180 ry 0 rz -180 deg; joints [-162.027, -45.478, -95.382, 22.697, 53.101, -14.097]
  Call Extruder(31984.19757)
  MoveL 3417 to (10.42, -8.31, 145) mm, rotated rx -180 ry 0 rz 180 deg; joints [-161.819, -45.675, -94.91, 23.03, 52.898, -14.383]
  Call Extruder(31988.86121)
  MoveL 3418 to (12.01, -5.78, 145) mm, rotated rx -180 ry 0 rz 180 deg; joints [-161.529, -45.847, -94.499, 23.454, 52.752, -14.714]
  Call Extruder(31993.52477)
  MoveL 3419 to (13, -2.97, 145) mm, rotated rx 180 ry 0 rz -180 deg; joints [-161.171, -45.985, -94.171, 23.947, 52.67, -15.073]
  Call Extruder(31998.18873)
  MoveL 3420 to (13.33, 0, 145) mm, rotated rx 180 ry 0 rz 180 deg; joints [-160.763, -46.082, -93.942, 24.484, 52.656, -15.442]
  Call Extruder(32002.85268)
  MoveL 3421 to (12.99, 2.97, 145) mm, rotated rx -180 ry 0 rz 180 deg; joints [-160.324, -46.132, -93.821, 25.038, 52.71, -15.801]
  Call Extruder(32007.51626)
  MoveL 3422 to (12.01, 5.78, 145) mm, rotated rx 180 ry 0 rz -180 deg; joints [-159.874, -46.135, -93.815, 25.582, 52.831, -16.132]
  Call Extruder(32012.17988)
  MoveL 3423 to (10.42, 8.31, 145) mm, rotated rx 180 ry 0 rz 180 deg; joints [-159.432, -46.089, -93.925, 26.092, 53.012, -16.417]
  Call Extruder(32016.84407)
  MoveL 3424 to (8.31, 10.42, 145) mm, rotated rx 180 ry 0 rz 180 deg; joints [-159.021, -45.996, -94.144, 26.544, 53.243, -16.643]
  Call Extruder(32021.50769)
  MoveL 3425 to (5.78, 12.01, 145) mm, rotated rx 180 ry 0 rz 180 deg; joints [-158.657, -45.863, -94.463, 26.916, 53.513, -16.798]
  Call Extruder(32026.17127)
  MoveL 3426 to (2.97, 12.99, 145) mm, rotated rx -180 ry 0 rz 180 deg; joints [-158.359, -45.694, -94.866, 27.191, 53.807, -16.876]
  Call Extruder(32030.83523)
  MoveL 3427 to (0, 13.33, 145) mm, rotated rx 180 ry 0 rz 180 deg; joints [-158.143, -45.499, -95.333, 27.357, 54.112, -16.872]
  Call Extruder(32035.49917)
  MoveL 3428 to (-2.97, 13, 145) mm, rotated rx 180 ry 0 rz 180 deg; joints [-158.019, -45.287, -95.843, 27.404, 54.412, -16.789]
  Call Extruder(32040.16274)
  MoveL 3429 to (-5.78, 12.01, 145) mm, rotated rx -180 ry 0 rz 180 deg; joints [-157.997, -45.069, -96.369, 27.329, 54.692, -16.63]
  Call Extruder(32044.82637)
  MoveL 3430 to (-8.31, 10.42, 145) mm, rotated rx -180 ry 0 rz 180 deg; joints [-158.08, -44.856, -96.886, 27.134, 54.939, -16.404]
  Call Extruder(32049.49056)
  MoveL 3431 to (-10.42, 8.31, 145) mm, rotated rx 180 ry 0 rz 180 deg; joints [-158.266, -44.658, -97.366, 26.826, 55.139, -16.122]
  Call Extruder(32054.15418)
  MoveL 3432 to (-12.01, 5.78, 145) mm, rotated rx 180 ry 0 rz 180 deg; joints [-158.549, -44.486, -97.787, 26.418, 55.284, -15.798]
  Call Extruder(32058.81776)
  MoveL 3433 to (-13, 2.97, 145) mm, rotated rx -180 ry 0 rz -180 deg; joints [-158.913, -44.348, -98.125, 25.93, 55.365, -15.448]
  Call Extruder(32063.48171)
  MoveL 3434 to (-13.33, 0, 145) mm, rotated rx 180 ry 0 rz 180 deg; joints [-159.341, -44.251, -98.363, 25.386, 55.38, -15.088]
  Call Extruder(32068.14567)
  MoveL 3435 to (-12.99, -2.97, 145) mm, rotated rx 180 ry 0 rz 180 deg; joints [-159.811, -44.2, -98.488, 24.813, 55.326, -14.736]
  Call Extruder(32072.80923)
  MoveL 3436 to (-12.01, -5.78, 145) mm, rotated rx -180 ry 0 rz 180 deg; joints [-160.294, -44.198, -98.494, 24.242, 55.208, -14.41]
  Call Extruder(32077.47286)
  MoveL 3437 to (-10.42, -8.31, 145) mm, rotated rx 180 ry 0 rz 180 deg; joints [-160.766, -44.244, -98.381, 23.703, 55.03, -14.124]
  Call Extruder(32082.13705)
  MoveL 3438 to (-8.31, -10.42, 145) mm, rotated rx -180 ry 0 rz 180 deg; joints [-161.2, -44.336, -98.153, 23.227, 54.801, -13.895]
  Call Extruder(32086.80068)
  MoveL 3439 to (-5.78, -12.01, 145) mm, rotated rx -180 ry 0 rz 180 deg; joints [-161.572, -44.471, -97.824, 22.839, 54.533, -13.732]
  Call Extruder(32091.46425)
  MoveL 3440 to (-2.97, -12.99, 145) mm, rotated rx 180 ry 0 rz 180 deg; joints [-161.863, -44.64, -97.411, 22.559, 54.239, -13.646]
  Call Extruder(32096.12820)
  MoveL 3441 to (0, -13.33, 145) mm, rotated rx 180 ry 0 rz -180 deg; joints [-162.059, -44.835, -96.935, 22.401, 53.933, -13.64]
  Call Extruder(32100.79215)
  MoveL 3442 to (2.97, -12.99, 145) mm, rotated rx -180 ry 0 rz -180 deg; joints [-162.152, -45.047, -96.421, 22.372, 53.632, -13.716]
  Set speed (130.0 mm/s)
  MoveL 3443 to (2.97, -12.99, 150) mm, rotated rx -180 ry 0 rz -180 deg; joints [-162.152, -44.302, -96.646, 22.52, 53.152, -13.963]
  MoveL 3444 to (-26.25, -4.54, 150) mm, rotated rx 180 ry 0 rz 180 deg; joints [-159.288, -42.519, -100.956, 25.197, 56.172, -14.678]
  Call Extruder(32103.02477)
  Set speed (60.0 mm/s)
  MoveL 3445 to (-26.09, -5.96, 150) mm, rotated rx 180 ry 0 rz 180 deg; joints [-159.522, -42.495, -101.016, 24.915, 56.145, -14.508]
  Call Extruder(32112.38956)
  MoveL 3446 to (-24.11, -11.61, 150) mm, rotated rx 180 ry 0 rz 180 deg; joints [-160.532, -42.49, -101.028, 23.733, 55.905, -13.845]
  Call Extruder(32121.75448)
  MoveL 3447 to (-20.93, -16.69, 150) mm, rotated rx 180 ry 0 rz 180 deg; joints [-161.513, -42.585, -100.794, 22.615, 55.547, -13.261]
  Call Extruder(32131.11969)
  MoveL 3448 to (-16.69, -20.93, 150) mm, rotated rx -180 ry 0 rz 180 deg; joints [-162.406, -42.775, -100.327, 21.629, 55.089, -12.785]
  Call Extruder(32140.48460)
  MoveL 3449 to (-11.61, -24.12, 150) mm, rotated rx 180 ry 0 rz 180 deg; joints [-163.159, -43.051, -99.654, 20.831, 54.554, -12.443]
  Call Extruder(32149.84940)
  MoveL 3450 to (-5.96, -26.09, 150) mm, rotated rx -180 ry 0 rz 180 deg; joints [-163.733, -43.398, -98.812, 20.266, 53.968, -12.254]
  Call Extruder(32159.21450)
  MoveL 3451 to (0, -26.77, 150) mm, rotated rx 180 ry 0 rz 180 deg; joints [-164.103, -43.799, -97.847, 19.96, 53.36, -12.229]
  Call Extruder(32168.57961)
  MoveL 3452 to (5.96, -26.09, 150) mm, rotated rx 180 ry 0 rz 180 deg; joints [-164.258, -44.234, -96.809, 19.925, 52.76, -12.373]
  Call Extruder(32177.94441)
  MoveL 3453 to (11.61, -24.11, 150) mm, rotated rx 180 ry 0 rz 180 deg; joints [-164.201, -44.68, -95.751, 20.156, 52.198, -12.68]
  Call Extruder(32187.30932)
  MoveL 3454 to (16.69, -20.93, 150) mm, rotated rx -180 ry 0 rz 180 deg; joints [-163.944, -45.116, -94.727, 20.635, 51.703, -13.136]
  Call Extruder(32196.67453)
  MoveL 3455 to (20.93, -16.69, 150) mm, rotated rx 180 ry 0 rz 180 deg; joints [-163.508, -45.519, -93.784, 21.331, 51.301, -13.72]
  Call Extruder(32206.03945)
  MoveL 3456 to (24.12, -11.61, 150) mm, rotated rx -180 ry 0 rz 180 deg; joints [-162.92, -45.87, -92.969, 22.202, 51.013, -14.401]
  Call Extruder(32215.40424)
  MoveL 3457 to (26.09, -5.96, 150) mm, rotated rx 180 ry 0 rz -180 deg; joints [-162.209, -46.151, -92.319, 23.202, 50.854, -15.142]
  Call Extruder(32224.76934)
  MoveL 3458 to (26.77, 0, 150) mm, rotated rx -180 ry 0 rz -180 deg; joints [-161.41, -46.348, -91.865, 24.279, 50.832, -15.903]
  Call Extruder(32234.13445)
  MoveL 3459 to (26.09, 5.96, 150) mm, rotated rx -180 ry 0 rz 180 deg; joints [-160.556, -46.452, -91.626, 25.382, 50.949, -16.642]
  Call Extruder(32243.49925)
  MoveL 3460 to (24.11, 11.61, 150) mm, rotated rx -180 ry 0 rz 180 deg; joints [-159.683, -46.457, -91.615, 26.458, 51.198, -17.32]
  Call Extruder(32252.86416)
  MoveL 3461 to (20.93, 16.69, 150) mm, rotated rx 180 ry 0 rz 180 deg; joints [-158.826, -46.363, -91.831, 27.459, 51.566, -17.902]
  Call Extruder(32262.22937)
  MoveL 3462 to (16.69, 20.93, 150) mm, rotated rx 180 ry 0 rz 180 deg; joints [-158.019, -46.174, -92.265, 28.344, 52.034, -18.359]
  Call Extruder(32271.59429)
  MoveL 3463 to (11.61, 24.11, 150) mm, rotated rx 180 ry 0 rz -180 deg; joints [-157.299, -45.901, -92.897, 29.074, 52.578, -18.669]
  Call Extruder(32280.95909)
  MoveL 3464 to (5.96, 26.09, 150) mm, rotated rx 180 ry 0 rz 180 deg; joints [-156.697, -45.557, -93.697, 29.62, 53.168, -18.82]
  Call Extruder(32290.32419)
  MoveL 3465 to (0, 26.77, 150) mm, rotated rx 180 ry 0 rz 180 deg; joints [-156.245, -45.158, -94.629, 29.957, 53.776, -18.808]
  Call Extruder(32299.68929)
  MoveL 3466 to (-5.96, 26.09, 150) mm, rotated rx 180 ry 0 rz -180 deg; joints [-155.969, -44.724, -95.647, 30.067, 54.372, -18.636]
  Call Extruder(32309.05409)
  MoveL 3467 to (-11.61, 24.11, 150) mm, rotated rx 180 ry 0 rz 180 deg; joints [-155.891, -44.278, -96.704, 29.941, 54.925, -18.314]
  Call Extruder(32318.41901)
  MoveL 3468 to (-16.69, 20.93, 150) mm, rotated rx 180 ry 0 rz -180 deg; joints [-156.025, -43.841, -97.746, 29.577, 55.409, -17.859]
  Call Extruder(32327.78421)
  MoveL 3469 to (-20.93, 16.69, 150) mm, rotated rx -180 ry 0 rz 180 deg; joints [-156.374, -43.436, -98.721, 28.984, 55.801, -17.294]
  Call Extruder(32337.14912)
  MoveL 3470 to (-24.11, 11.61, 150) mm, rotated rx -180 ry 0 rz 180 deg; joints [-156.928, -43.083, -99.577, 28.181, 56.081, -16.645]
  Call Extruder(32346.51393)
  MoveL 3471 to (-26.09, 5.96, 150) mm, rotated rx -180 ry 0 rz 180 deg; joints [-157.665, -42.799, -100.269, 27.202, 56.235, -15.942]
  Call Extruder(32355.87903)
  MoveL 3472 to (-26.77, 0, 150) mm, rotated rx 180 ry 0 rz 180 deg; joints [-158.546, -42.6, -100.758, 26.094, 56.257, -15.219]
  Call Extruder(32360.66777)
  MoveL 3473 to (-26.42, -3.05, 150) mm, rotated rx 180 ry 0 rz 180 deg; joints [-159.044, -42.545, -100.892, 25.493, 56.2, -14.856]
  Set speed (130.0 mm/s)
  MoveL 3474 to (-41.86, -6.3, 150) mm, rotated rx 180 ry 0 rz 180 deg; joints [-158.606, -41.483, -103.539, 25.555, 57.74, -14.317]
  Call Extruder(32365.66561)
  Set speed (60.0 mm/s)
  MoveL 3475 to (-41.51, -9.47, 150) mm, rotated rx 180 ry 0 rz 180 deg; joints [-159.151, -41.429, -103.676, 24.906, 57.682, -13.941]
  Call Extruder(32380.56126)
  MoveL 3476 to (-38.36, -18.47, 150) mm, rotated rx 180 ry 0 rz 180 deg; joints [-160.835, -41.421, -103.696, 22.961, 57.302, -12.891]
  Call Extruder(32395.45712)
  MoveL 3477 to (-33.28, -26.54, 150) mm, rotated rx 180 ry 0 rz 180 deg; joints [-162.466, -41.573, -103.313, 21.119, 56.737, -11.961]
  Call Extruder(32410.35293)
  MoveL 3478 to (-26.54, -33.28, 150) mm, rotated rx 180 ry 0 rz -180 deg; joints [-163.93, -41.877, -102.55, 19.503, 56.013, -11.199]
  Call Extruder(32425.24879)
  MoveL 3479 to (-18.47, -38.36, 150) mm, rotated rx -180 ry 0 rz 180 deg; joints [-165.137, -42.316, -101.456, 18.211, 55.165, -10.643]
  Call Extruder(32440.14444)
  MoveL 3480 to (-9.47, -41.5, 150) mm, rotated rx 180 ry 0 rz 180 deg; joints [-166.024, -42.87, -100.096, 17.316, 54.235, -10.327]
  Call Extruder(32455.04031)
  MoveL 3481 to (0, -42.57, 150) mm, rotated rx 180 ry 0 rz 180 deg; joints [-166.562, -43.509, -98.545, 16.856, 53.268, -10.271]
  Call Extruder(32469.93618)
  MoveL 3482 to (9.47, -41.51, 150) mm, rotated rx -180 ry 0 rz 180 deg; joints [-166.745, -44.201, -96.889, 16.843, 52.311, -10.486]
  Call Extruder(32484.83185)
  MoveL 3483 to (18.47, -38.36, 150) mm, rotated rx -180 ry 0 rz 180 deg; joints [-166.591, -44.91, -95.21, 17.258, 51.413, -10.966]
  Call Extruder(32499.72769)
  MoveL 3484 to (26.54, -33.28, 150) mm, rotated rx 180 ry 0 rz -180 deg; joints [-166.133, -45.602, -93.591, 18.064, 50.62, -11.692]
  Call Extruder(32514.62351)
  MoveL 3485 to (33.29, -26.54, 150) mm, rotated rx 180 ry 0 rz 180 deg; joints [-165.409, -46.243, -92.107, 19.207, 49.973, -12.629]
  Call Extruder(32529.51936)
  MoveL 3486 to (38.36, -18.47, 150) mm, rotated rx 180 ry 0 rz 180 deg; joints [-164.468, -46.8, -90.828, 20.617, 49.509, -13.728]
  Call Extruder(32544.41501)
  MoveL 3487 to (41.5, -9.47, 150) mm, rotated rx -180 ry 0 rz 180 deg; joints [-163.355, -47.246, -89.81, 22.216, 49.251, -14.928]
  Call Extruder(32559.31089)
  MoveL 3488 to (42.57, 0, 150) mm, rotated rx 180 ry 0 rz 180 deg; joints [-162.12, -47.559, -89.099, 23.922, 49.216, -16.159]
  Call Extruder(32574.20676)
  MoveL 3489 to (41.5, 9.47, 150) mm, rotated rx -180 ry 0 rz 180 deg; joints [-160.81, -47.723, -88.726, 25.65, 49.405, -17.353]
  Call Extruder(32589.10243)
  MoveL 3490 to (38.36, 18.47, 150) mm, rotated rx 180 ry 0 rz 180 deg; joints [-159.475, -47.731, -88.708, 27.323, 49.806, -18.44]
  Call Extruder(32603.99827)
  MoveL 3491 to (33.29, 26.54, 150) mm, rotated rx 180 ry 0 rz 180 deg; joints [-158.16, -47.582, -89.046, 28.869, 50.398, -19.364]
  Call Extruder(32618.89409)
  MoveL 3492 to (26.54, 33.28, 150) mm, rotated rx -180 ry 0 rz 180 deg; joints [-156.916, -47.283, -89.725, 30.229, 51.149, -20.078]
  Call Extruder(32633.78994)
  MoveL 3493 to (18.47, 38.36, 150) mm, rotated rx -180 ry 0 rz -180 deg; joints [-155.789, -46.849, -90.714, 31.352, 52.018, -20.554]
  Call Extruder(32648.68560)
  MoveL 3494 to (9.47, 41.51, 150) mm, rotated rx -180 ry 0 rz -180 deg; joints [-154.828, -46.302, -91.97, 32.199, 52.959, -20.773]
  Call Extruder(32663.58147)
  MoveL 3495 to (0, 42.57, 150) mm, rotated rx -180 ry 0 rz 180 deg; joints [-154.081, -45.669, -93.436, 32.737, 53.926, -20.735]
  Call Extruder(32678.47735)
  MoveL 3496 to (-9.47, 41.51, 150) mm, rotated rx -180 ry 0 rz 180 deg; joints [-153.594, -44.98, -95.045, 32.941, 54.871, -20.447]
  Call Extruder(32693.37300)
  MoveL 3497 to (-18.47, 38.36, 150) mm, rotated rx -180 ry 0 rz 180 deg; joints [-153.408, -44.271, -96.722, 32.789, 55.747, -19.93]
  Call Extruder(32708.26885)
  MoveL 3498 to (-26.54, 33.28, 150) mm, rotated rx 180 ry 0 rz 180 deg; joints [-153.557, -43.576, -98.384, 32.271, 56.513, -19.209]
  Call Extruder(32723.16467)
  MoveL 3499 to (-33.29, 26.54, 150) mm, rotated rx 180 ry 0 rz 180 deg; joints [-154.059, -42.93, -99.949, 31.386, 57.133, -18.319]
  Call Extruder(32738.06051)
  MoveL 3500 to (-38.36, 18.47, 150) mm, rotated rx 180 ry 0 rz 180 deg; joints [-154.913, -42.367, -101.332, 30.152, 57.576, -17.3]
  Call Extruder(32752.95617)
  MoveL 3501 to (-41.51, 9.47, 150) mm, rotated rx 180 ry 0 rz 180 deg; joints [-156.091, -41.914, -102.456, 28.61, 57.822, -16.197]
  Call Extruder(32767.85205)
  MoveL 3502 to (-42.57, 0, 150) mm, rotated rx 180 ry 0 rz -180 deg; joints [-157.533, -41.596, -103.253, 26.829, 57.858, -15.061]
  Call Extruder(32775.40633)
  MoveL 3503 to (-42.03, -4.8, 150) mm, rotated rx -180 ry 0 rz 180 deg; joints [-158.35, -41.509, -103.473, 25.858, 57.768, -14.493]
  Set speed (130.0 mm/s)
  MoveL 3504 to (-54.1, -7.67, 150) mm, rotated rx -180 ry 0 rz 180 deg; joints [-158.024, -40.704, -105.53, 25.893, 58.974, -14.047]
  Call Extruder(32779.47896)
  Set speed (30.0 mm/s)
  MoveL 3505 to (-53.59, -12.23, 150) mm, rotated rx 180 ry 0 rz 180 deg; joints [-158.835, -40.627, -105.729, 24.942, 58.892, -13.511]
  Call Extruder(32790.40909)
  MoveL 3506 to (-49.52, -23.85, 150) mm, rotated rx -180 ry 0 rz 180 deg; joints [-161.095, -40.616, -105.756, 22.357, 58.404, -12.161]
  Call Extruder(32801.33938)
  MoveL 3507 to (-42.98, -34.27, 150) mm, rotated rx 180 ry 0 rz 180 deg; joints [-163.275, -40.813, -105.249, 19.91, 57.677, -10.96]
  Call Extruder(32812.26949)
  MoveL 3508 to (-34.27, -42.98, 150) mm, rotated rx 180 ry 0 rz 180 deg; joints [-165.21, -41.206, -104.243, 17.774, 56.745, -9.97]
  Call Extruder(32823.19978)
  MoveL 3509 to (-23.85, -49.52, 150) mm, rotated rx 180 ry 0 rz 180 deg; joints [-166.774, -41.775, -102.805, 16.088, 55.654, -9.242]
  Call Extruder(32834.12991)
  MoveL 3510 to (-12.23, -53.59, 150) mm, rotated rx 180 ry 0 rz 180 deg; joints [-167.889, -42.491, -101.026, 14.943, 54.454, -8.819]
  Call Extruder(32845.06013)
  MoveL 3511 to (0, -54.97, 150) mm, rotated rx 180 ry 0 rz 180 deg; joints [-168.526, -43.317, -99.01, 14.383, 53.206, -8.732]
  Call Extruder(32855.55849)
  MoveL 3512 to (11.75, -53.64, 150) mm, rotated rx 180 ry 0 rz 180 deg; joints [-168.69, -44.174, -96.952, 14.407, 52.017, -8.984]
  Call Extruder(32855.99035)
  MoveL 3513 to (12.23, -53.59, 150) mm, rotated rx -180 ry 0 rz 180 deg; joints [-168.697, -44.21, -96.866, 14.409, 51.968, -8.995]
  Call Extruder(32866.92050)
  MoveL 3514 to (23.85, -49.53, 150) mm, rotated rx -180 ry 0 rz 180 deg; joints [-168.436, -45.126, -94.704, 14.99, 50.804, -9.605]
  Call Extruder(32877.85078)
  MoveL 3515 to (34.27, -42.98, 150) mm, rotated rx 180 ry 0 rz 180 deg; joints [-167.797, -46.019, -92.625, 16.073, 49.773, -10.54]
  Call Extruder(32888.78090)
  MoveL 3516 to (42.98, -34.27, 150) mm, rotated rx -180 ry 0 rz 180 deg; joints [-166.837, -46.845, -90.725, 17.58, 48.931, -11.759]
  Call Extruder(32899.71118)
  MoveL 3517 to (49.52, -23.85, 150) mm, rotated rx -180 ry 0 rz 180 deg; joints [-165.618, -47.563, -89.089, 19.423, 48.324, -13.195]
  Call Extruder(32910.64131)
  MoveL 3518 to (53.59, -12.23, 150) mm, rotated rx -180 ry 0 rz -180 deg; joints [-164.2, -48.139, -87.789, 21.497, 47.988, -14.768]
  Call Extruder(32921.57153)
  MoveL 3519 to (54.97, 0, 150) mm, rotated rx -180 ry 0 rz 180 deg; joints [-162.641, -48.542, -86.881, 23.695, 47.941, -16.383]
  Call Extruder(32932.50176)
  MoveL 3520 to (53.59, 12.23, 150) mm, rotated rx 180 ry 0 rz 180 deg; joints [-160.996, -48.755, -86.405, 25.906, 48.187, -17.943]
  Call Extruder(32943.43190)
  MoveL 3521 to (49.52, 23.85, 150) mm, rotated rx 180 ry 0 rz -180 deg; joints [-159.322, -48.765, -86.382, 28.031, 48.711, -19.356]
  Call Extruder(32954.36218)
  MoveL 3522 to (42.98, 34.27, 150) mm, rotated rx 180 ry 0 rz 180 deg; joints [-157.673, -48.572, -86.814, 29.982, 49.483, -20.547]
  Call Extruder(32965.29230)
  MoveL 3523 to (34.27, 42.98, 150) mm, rotated rx -180 ry 0 rz 180 deg; joints [-156.102, -48.187, -87.68, 31.689, 50.459, -21.456]
  Call Extruder(32976.22258)
  MoveL 3524 to (23.85, 49.52, 150) mm, rotated rx -180 ry 0 rz 180 deg; joints [-154.667, -47.627, -88.944, 33.099, 51.585, -22.049]
  Call Extruder(32987.15272)
  MoveL 3525 to (12.23, 53.59, 150) mm, rotated rx 180 ry 0 rz 180 deg; joints [-153.426, -46.921, -90.549, 34.167, 52.803, -22.31]
  Call Extruder(32998.08294)
  MoveL 3526 to (0, 54.97, 150) mm, rotated rx -180 ry 0 rz 180 deg; joints [-152.438, -46.104, -92.427, 34.86, 54.051, -22.241]
  Call Extruder(33009.01316)
  MoveL 3527 to (-12.23, 53.59, 150) mm, rotated rx 180 ry 0 rz 180 deg; joints [-151.764, -45.216, -94.492, 35.147, 55.269, -21.856]
  Call Extruder(33019.94330)
  MoveL 3528 to (-23.85, 49.52, 150) mm, rotated rx 180 ry 0 rz 180 deg; joints [-151.463, -44.3, -96.651, 35, 56.396, -21.182]
  Call Extruder(33030.87358)
  MoveL 3529 to (-34.27, 42.98, 150) mm, rotated rx 180 ry 0 rz 180 deg; joints [-151.589, -43.403, -98.801, 34.394, 57.382, -20.254]
  Call Extruder(33041.80370)
  MoveL 3530 to (-42.98, 34.27, 150) mm, rotated rx -180 ry 0 rz -180 deg; joints [-152.179, -42.568, -100.835, 33.316, 58.179, -19.114]
  Call Extruder(33052.73398)
  MoveL 3531 to (-49.52, 23.85, 150) mm, rotated rx 180 ry 0 rz -180 deg; joints [-153.248, -41.84, -102.642, 31.771, 58.75, -17.812]
  Call Extruder(33063.66412)
  MoveL 3532 to (-53.59, 12.23, 150) mm, rotated rx -180 ry 0 rz -180 deg; joints [-154.769, -41.255, -104.118, 29.798, 59.068, -16.402]
  Call Extruder(33074.59434)
  MoveL 3533 to (-54.97, 0, 150) mm, rotated rx 180 ry 0 rz -180 deg; joints [-156.673, -40.843, -105.17, 27.478, 59.116, -14.947]
  Call Extruder(33080.11996)
  MoveL 3534 to (-54.27, -6.18, 150) mm, rotated rx -180 ry 0 rz 180 deg; joints [-157.76, -40.73, -105.462, 26.203, 59.002, -14.222]
  Set speed (130.0 mm/s)
  MoveL 3535 to (-49.9, -9.51, 150) mm, rotated rx 180 ry 0 rz 180 deg; joints [-158.616, -40.913, -104.991, 25.307, 58.534, -13.865]
  MoveL 3536 to (-4.91, 13.82, 150) mm, rotated rx 180 ry 0 rz 180 deg; joints [-157.786, -44.435, -96.332, 27.799, 54.159, -17.156]
  Call Extruder(33113.29496)
  Set speed (20.0 mm/s)
  MoveL 3537 to (-13.82, 4.92, 150) mm, rotated rx 180 ry 0 rz 180 deg; joints [-158.572, -43.585, -98.363, 26.491, 54.986, -15.959]
  Call Extruder(33183.10157)
  MoveL 3538 to (4.91, -13.82, 150) mm, rotated rx -180 ry 0 rz 180 deg; joints [-162.368, -44.422, -96.363, 22.305, 52.948, -13.884]
  Call Extruder(33216.27659)
  MoveL 3539 to (13.82, -4.91, 150) mm, rotated rx 180 ry 0 rz 180 deg; joints [-161.491, -45.27, -94.366, 23.719, 52.11, -15.101]
  Set speed (130.0 mm/s)
  MoveL 3540 to (13.82, -4.91, 155) mm, rotated rx 180 ry 0 rz 180 deg; joints [-161.491, -44.546, -94.579, 23.881, 51.643, -15.363]
  MoveL 3541 to (-26.25, -4.54, 155) mm, rotated rx -180 ry 0 rz 180 deg; joints [-159.288, -41.739, -101.178, 25.359, 55.666, -14.966]
  Call Extruder(33218.50920)
  Set speed (60.0 mm/s)
  MoveL 3542 to (-26.09, -5.96, 155) mm, rotated rx 180 ry 0 rz 180 deg; joints [-159.522, -41.714, -101.238, 25.075, 55.638, -14.794]
  Call Extruder(33227.87399)
  MoveL 3543 to (-24.11, -11.61, 155) mm, rotated rx -180 ry 0 rz 180 deg; joints [-160.532, -41.709, -101.25, 23.887, 55.393, -14.119]
  Call Extruder(33237.23891)
  MoveL 3544 to (-20.93, -16.69, 155) mm, rotated rx 180 ry 0 rz 180 deg; joints [-161.513, -41.806, -101.016, 22.764, 55.032, -13.522]
  Call Extruder(33246.60412)
  MoveL 3545 to (-16.69, -20.93, 155) mm, rotated rx 180 ry 0 rz 180 deg; joints [-162.406, -42.001, -100.548, 21.773, 54.575, -13.036]
  Call Extruder(33255.96904)
  MoveL 3546 to (-11.61, -24.12, 155) mm, rotated rx -180 ry 0 rz 180 deg; joints [-163.159, -42.283, -99.874, 20.972, 54.042, -12.684]
  Call Extruder(33265.33383)
  MoveL 3547 to (-5.96, -26.09, 155) mm, rotated rx 180 ry 0 rz 180 deg; joints [-163.733, -42.637, -99.031, 20.404, 53.46, -12.488]
  Call Extruder(33274.69893)
  MoveL 3548 to (0, -26.77, 155) mm, rotated rx 180 ry 0 rz 180 deg; joints [-164.103, -43.047, -98.064, 20.097, 52.857, -12.458]
  Call Extruder(33284.06403)
  MoveL 3549 to (5.96, -26.09, 155) mm, rotated rx -180 ry 0 rz 180 deg; joints [-164.258, -43.49, -97.024, 20.064, 52.264, -12.6]
  Call Extruder(33293.42884)
  MoveL 3550 to (11.61, -24.11, 155) mm, rotated rx -180 ry 0 rz 180 deg; joints [-164.201, -43.945, -95.966, 20.297, 51.709, -12.908]
  Call Extruder(33302.79375)
  MoveL 3551 to (16.69, -20.93, 155) mm, rotated rx -180 ry 0 rz 180 deg; joints [-163.944, -44.389, -94.94, 20.78, 51.223, -13.369]
  Call Extruder(33312.15896)
  MoveL 3552 to (20.93, -16.69, 155) mm, rotated rx 180 ry 0 rz -180 deg; joints [-163.508, -44.8, -93.996, 21.48, 50.829, -13.958]
  Call Extruder(33321.52388)
  MoveL 3553 to (24.12, -11.61, 155) mm, rotated rx 180 ry 0 rz 180 deg; joints [-162.92, -45.156, -93.18, 22.357, 50.548, -14.647]
  Call Extruder(33330.88867)
  MoveL 3554 to (26.09, -5.96, 155) mm, rotated rx 180 ry 0 rz -180 deg; joints [-162.209, -45.442, -92.53, 23.364, 50.396, -15.397]
  Call Extruder(33340.25377)
  MoveL 3555 to (26.77, 0, 155) mm, rotated rx 180 ry 0 rz -180 deg; joints [-161.41, -45.643, -92.075, 24.447, 50.38, -16.167]
  Call Extruder(33349.61888)
  MoveL 3556 to (26.09, 5.96, 155) mm, rotated rx 180 ry 0 rz 180 deg; joints [-160.556, -45.748, -91.836, 25.556, 50.503, -16.916]
  Call Extruder(33358.98368)
  MoveL 3557 to (24.12, 11.61, 155) mm, rotated rx 180 ry 0 rz 180 deg; joints [-159.683, -45.753, -91.825, 26.637, 50.756, -17.604]
  Call Extruder(33368.34859)
  MoveL 3558 to (20.93, 16.69, 155) mm, rotated rx -180 ry 0 rz -180 deg; joints [-158.826, -45.657, -92.041, 27.643, 51.127, -18.195]
  Call Extruder(33377.71380)
  MoveL 3559 to (16.69, 20.93, 155) mm, rotated rx -180 ry 0 rz 180 deg; joints [-158.019, -45.466, -92.475, 28.53, 51.596, -18.66]
  Call Extruder(33387.07871)
  MoveL 3560 to (11.61, 24.11, 155) mm, rotated rx 180 ry 0 rz 180 deg; joints [-157.299, -45.188, -93.108, 29.263, 52.139, -18.978]
  Call Extruder(33396.44352)
  MoveL 3561 to (5.96, 26.09, 155) mm, rotated rx 180 ry 0 rz 180 deg; joints [-156.697, -44.838, -93.909, 29.81, 52.728, -19.135]
  Call Extruder(33405.80862)
  MoveL 3562 to (0, 26.77, 155) mm, rotated rx 180 ry 0 rz 180 deg; joints [-156.245, -44.432, -94.842, 30.146, 53.332, -19.127]
  Call Extruder(33415.17372)
  MoveL 3563 to (-5.96, 26.09, 155) mm, rotated rx -180 ry 0 rz 180 deg; joints [-155.969, -43.99, -95.862, 30.256, 53.922, -18.958]
  Call Extruder(33424.53852)
  MoveL 3564 to (-11.61, 24.11, 155) mm, rotated rx 180 ry 0 rz -180 deg; joints [-155.891, -43.535, -96.919, 30.128, 54.469, -18.637]
  Call Extruder(33433.90344)
  MoveL 3565 to (-16.69, 20.93, 155) mm, rotated rx 180 ry 0 rz -180 deg; joints [-156.025, -43.09, -97.963, 29.761, 54.945, -18.182]
  Call Extruder(33443.26864)
  MoveL 3566 to (-20.93, 16.69, 155) mm, rotated rx 180 ry 0 rz -180 deg; joints [-156.374, -42.676, -98.939, 29.164, 55.327, -17.613]
  Call Extruder(33452.63356)
  MoveL 3567 to (-24.12, 11.61, 155) mm, rotated rx 180 ry 0 rz 180 deg; joints [-156.928, -42.315, -99.797, 28.357, 55.598, -16.959]
  Call Extruder(33461.99835)
  MoveL 3568 to (-26.09, 5.96, 155) mm, rotated rx 180 ry 0 rz -180 deg; joints [-157.665, -42.025, -100.49, 27.373, 55.743, -16.249]
  Call Extruder(33471.36346)
  MoveL 3569 to (-26.77, 0, 155) mm, rotated rx 180 ry 0 rz 180 deg; joints [-158.546, -41.821, -100.98, 26.26, 55.757, -15.515]
  Call Extruder(33476.15220)
  MoveL 3570 to (-26.42, -3.05, 155) mm, rotated rx 180 ry 0 rz 180 deg; joints [-159.044, -41.765, -101.114, 25.656, 55.696, -15.147]
  Set speed (130.0 mm/s)
  MoveL 3571 to (-41.86, -6.3, 155) mm, rotated rx -180 ry 0 rz 180 deg; joints [-158.606, -40.676, -103.766, 25.715, 57.218, -14.615]
  Call Extruder(33481.15004)
  Set speed (60.0 mm/s)
  MoveL 3572 to (-41.5, -9.47, 155) mm, rotated rx 180 ry 0 rz 180 deg; joints [-159.151, -40.621, -103.903, 25.063, 57.155, -14.232]
  Call Extruder(33496.04569)
  MoveL 3573 to (-38.36, -18.47, 155) mm, rotated rx 180 ry 0 rz 180 deg; joints [-160.835, -40.613, -103.923, 23.108, 56.767, -13.162]
  Call Extruder(33510.94155)
  MoveL 3574 to (-33.28, -26.54, 155) mm, rotated rx 180 ry 0 rz 180 deg; joints [-162.466, -40.769, -103.539, 21.258, 56.198, -12.212]
  Call Extruder(33525.83736)
  MoveL 3575 to (-26.54, -33.28, 155) mm, rotated rx 180 ry 0 rz -180 deg; joints [-163.93, -41.08, -102.775, 19.633, 55.474, -11.43]
  Call Extruder(33540.73322)
  MoveL 3576 to (-18.47, -38.36, 155) mm, rotated rx -180 ry 0 rz 180 deg; joints [-165.137, -41.531, -101.679, 18.335, 54.631, -10.859]
  Call Extruder(33555.62886)
  MoveL 3577 to (-9.47, -41.51, 155) mm, rotated rx 180 ry 0 rz 180 deg; joints [-166.024, -42.097, -100.316, 17.436, 53.708, -10.531]
  Call Extruder(33570.52474)
  MoveL 3578 to (0, -42.57, 155) mm, rotated rx 180 ry 0 rz -180 deg; joints [-166.562, -42.75, -98.763, 16.975, 52.75, -10.468]
  Call Extruder(33585.42061)
  MoveL 3579 to (9.47, -41.51, 155) mm, rotated rx -180 ry 0 rz 180 deg; joints [-166.745, -43.456, -97.104, 16.962, 51.805, -10.681]
  Call Extruder(33600.31627)
  MoveL 3580 to (18.47, -38.36, 155) mm, rotated rx 180 ry 0 rz -180 deg; joints [-166.591, -44.18, -95.423, 17.382, 50.919, -11.163]
  Call Extruder(33615.21212)
  MoveL 3581 to (26.54, -33.28, 155) mm, rotated rx 180 ry 0 rz 180 deg; joints [-166.133, -44.884, -93.802, 18.195, 50.138, -11.896]
  Call Extruder(33630.10794)
  MoveL 3582 to (33.29, -26.54, 155) mm, rotated rx -180 ry 0 rz 180 deg; joints [-165.409, -45.535, -92.318, 19.346, 49.504, -12.844]
  Call Extruder(33645.00379)
  MoveL 3583 to (38.36, -18.47, 155) mm, rotated rx -180 ry 0 rz 180 deg; joints [-164.468, -46.101, -91.037, 20.765, 49.051, -13.956]
  Call Extruder(33659.89944)
  MoveL 3584 to (41.51, -9.47, 155) mm, rotated rx 180 ry 0 rz 180 deg; joints [-163.355, -46.554, -90.018, 22.375, 48.804, -15.17]
  Call Extruder(33674.79532)
  MoveL 3585 to (42.57, 0, 155) mm, rotated rx 180 ry 0 rz 180 deg; joints [-162.12, -46.872, -89.306, 24.091, 48.778, -16.418]
  Call Extruder(33689.69119)
  MoveL 3586 to (41.5, 9.47, 155) mm, rotated rx 180 ry 0 rz 180 deg; joints [-160.81, -47.039, -88.933, 25.829, 48.975, -17.626]
  Call Extruder(33704.58685)
  MoveL 3587 to (38.36, 18.47, 155) mm, rotated rx 180 ry 0 rz 180 deg; joints [-159.475, -47.047, -88.915, 27.51, 49.383, -18.728]
  Call Extruder(33719.48270)
  MoveL 3588 to (33.29, 26.54, 155) mm, rotated rx 180 ry 0 rz 180 deg; joints [-158.16, -46.896, -89.254, 29.063, 49.98, -19.666]
  Call Extruder(33734.37852)
  MoveL 3589 to (26.54, 33.28, 155) mm, rotated rx 180 ry 0 rz 180 deg; joints [-156.916, -46.592, -89.933, 30.427, 50.732, -20.392]
  Call Extruder(33749.27436)
  MoveL 3590 to (18.47, 38.36, 155) mm, rotated rx -180 ry 0 rz -180 deg; joints [-155.789, -46.152, -90.923, 31.553, 51.601, -20.878]
  Call Extruder(33764.17003)
  MoveL 3591 to (9.47, 41.51, 155) mm, rotated rx -180 ry 0 rz 180 deg; joints [-154.828, -45.596, -92.18, 32.401, 52.54, -21.106]
  Call Extruder(33779.06590)
  MoveL 3592 to (0, 42.57, 155) mm, rotated rx -180 ry 0 rz 180 deg; joints [-154.081, -44.952, -93.648, 32.939, 53.502, -21.075]
  Call Extruder(33793.96177)
  MoveL 3593 to (-9.47, 41.5, 155) mm, rotated rx 180 ry 0 rz 180 deg; joints [-153.594, -44.251, -95.258, 33.14, 54.438, -20.792]
  Call Extruder(33808.85742)
  MoveL 3594 to (-18.47, 38.36, 155) mm, rotated rx 180 ry 0 rz 180 deg; joints [-153.408, -43.528, -96.937, 32.986, 55.304, -20.277]
  Call Extruder(33823.75328)
  MoveL 3595 to (-26.54, 33.29, 155) mm, rotated rx 180 ry 0 rz 180 deg; joints [-153.557, -42.819, -98.602, 32.464, 56.058, -19.556]
  Call Extruder(33838.64909)
  MoveL 3596 to (-33.28, 26.54, 155) mm, rotated rx 180 ry 0 rz 180 deg; joints [-154.059, -42.159, -100.169, 31.574, 56.663, -18.662]
  Call Extruder(33853.54494)
  MoveL 3597 to (-38.36, 18.47, 155) mm, rotated rx -180 ry 0 rz 180 deg; joints [-154.913, -41.582, -101.555, 30.334, 57.091, -17.636]
  Call Extruder(33868.44060)
  MoveL 3598 to (-41.5, 9.47, 155) mm, rotated rx 180 ry 0 rz 180 deg; joints [-156.091, -41.119, -102.68, 28.784, 57.321, -16.522]
  Call Extruder(33883.33648)
  MoveL 3599 to (-42.57, 0, 155) mm, rotated rx -180 ry 0 rz -180 deg; joints [-157.533, -40.793, -103.48, 26.995, 57.343, -15.37]
  Call Extruder(33890.89076)
  MoveL 3600 to (-42.03, -4.8, 155) mm, rotated rx -180 ry 0 rz 180 deg; joints [-158.35, -40.703, -103.7, 26.019, 57.247, -14.794]
  Set speed (130.0 mm/s)
  MoveL 3601 to (-54.1, -7.67, 155) mm, rotated rx 180 ry 0 rz 180 deg; joints [-158.024, -39.875, -105.761, 26.052, 58.437, -14.353]
  Call Extruder(33894.96339)
  Set speed (30.0 mm/s)
  MoveL 3602 to (-53.59, -12.23, 155) mm, rotated rx 180 ry 0 rz 180 deg; joints [-158.835, -39.796, -105.96, 25.096, 58.348, -13.808]
  Call Extruder(33905.89352)
  MoveL 3603 to (-49.53, -23.85, 155) mm, rotated rx 180 ry 0 rz 180 deg; joints [-161.095, -39.786, -105.987, 22.5, 57.85, -12.43]
  Call Extruder(33916.82381)
  MoveL 3604 to (-42.98, -34.27, 155) mm, rotated rx 180 ry 0 rz 180 deg; joints [-163.275, -39.988, -105.479, 20.04, 57.118, -11.202]
  Call Extruder(33927.75392)
  MoveL 3605 to (-34.27, -42.98, 155) mm, rotated rx -180 ry 0 rz 180 deg; joints [-165.21, -40.392, -104.471, 17.893, 56.188, -10.185]
  Call Extruder(33938.68421)
  MoveL 3606 to (-23.85, -49.53, 155) mm, rotated rx 180 ry 0 rz 180 deg; joints [-166.774, -40.976, -103.03, 16.198, 55.102, -9.436]
  Call Extruder(33949.61434)
  MoveL 3607 to (-12.23, -53.59, 155) mm, rotated rx 180 ry 0 rz 180 deg; joints [-167.889, -41.709, -101.248, 15.048, 53.914, -8.998]
  Call Extruder(33960.54456)
  MoveL 3608 to (0, -54.97, 155) mm, rotated rx -180 ry 0 rz 180 deg; joints [-168.526, -42.554, -99.229, 14.485, 52.679, -8.902]
  Call Extruder(33971.47478)
  MoveL 3609 to (12.23, -53.59, 155) mm, rotated rx 180 ry 0 rz 180 deg; joints [-168.697, -43.466, -97.082, 14.513, 51.457, -9.163]
  Call Extruder(33982.40492)
  MoveL 3610 to (23.85, -49.53, 155) mm, rotated rx 180 ry 0 rz 180 deg; joints [-168.436, -44.399, -94.917, 15.1, 50.308, -9.777]
  Call Extruder(33993.33520)
  MoveL 3611 to (34.27, -42.98, 155) mm, rotated rx -180 ry 0 rz 180 deg; joints [-167.797, -45.308, -92.835, 16.191, 49.293, -10.723]
  Call Extruder(34004.26532)
  MoveL 3612 to (42.98, -34.27, 155) mm, rotated rx 180 ry 0 rz 180 deg; joints [-166.837, -46.147, -90.934, 17.711, 48.465, -11.956]
  Call Extruder(34015.19561)
  MoveL 3613 to (49.52, -23.85, 155) mm, rotated rx 180 ry 0 rz 180 deg; joints [-165.618, -46.876, -89.297, 19.566, 47.873, -13.41]
  Call Extruder(34026.12574)
  MoveL 3614 to (53.59, -12.23, 155) mm, rotated rx 180 ry 0 rz -180 deg; joints [-164.2, -47.46, -87.995, 21.655, 47.549, -15.002]
  Call Extruder(34037.05596)
  MoveL 3615 to (54.97, 0, 155) mm, rotated rx 180 ry 0 rz 180 deg; joints [-162.641, -47.87, -87.087, 23.866, 47.514, -16.637]
  Call Extruder(34047.98618)
  MoveL 3616 to (53.59, 12.23, 155) mm, rotated rx 180 ry 0 rz 180 deg; joints [-160.996, -48.085, -86.611, 26.089, 47.77, -18.217]
  Call Extruder(34058.91633)
  MoveL 3617 to (49.52, 23.85, 155) mm, rotated rx 180 ry 0 rz -180 deg; joints [-159.322, -48.095, -86.588, 28.224, 48.302, -19.648]
  Call Extruder(34069.84660)
  MoveL 3618 to (42.98, 34.27, 155) mm, rotated rx 180 ry 0 rz 180 deg; joints [-157.673, -47.9, -87.02, 30.183, 49.08, -20.855]
  Call Extruder(34080.77673)
  MoveL 3619 to (34.27, 42.98, 155) mm, rotated rx 180 ry 0 rz -180 deg; joints [-156.102, -47.509, -87.887, 31.896, 50.059, -21.779]
  Call Extruder(34091.70700)
  MoveL 3620 to (23.85, 49.52, 155) mm, rotated rx -180 ry 0 rz 180 deg; joints [-154.667, -46.941, -89.151, 33.308, 51.185, -22.385]
  Call Extruder(34102.63715)
  MoveL 3621 to (12.23, 53.59, 155) mm, rotated rx 180 ry 0 rz -180 deg; joints [-153.426, -46.225, -90.758, 34.377, 52.4, -22.656]
  Call Extruder(34113.56737)
  MoveL 3622 to (0, 54.97, 155) mm, rotated rx 180 ry 0 rz 180 deg; joints [-152.438, -45.395, -92.637, 35.069, 53.642, -22.595]
  Call Extruder(34124.49759)
  MoveL 3623 to (-12.23, 53.59, 155) mm, rotated rx 180 ry 0 rz 180 deg; joints [-151.764, -44.491, -94.705, 35.353, 54.85, -22.217]
  Call Extruder(34135.42773)
  MoveL 3624 to (-23.85, 49.52, 155) mm, rotated rx -180 ry 0 rz 180 deg; joints [-151.463, -43.558, -96.866, 35.203, 55.965, -21.547]
  Call Extruder(34146.35801)
  MoveL 3625 to (-34.27, 42.98, 155) mm, rotated rx 180 ry 0 rz 180 deg; joints [-151.589, -42.642, -99.02, 34.592, 56.935, -20.62]
  Call Extruder(34157.28813)
  MoveL 3626 to (-42.98, 34.27, 155) mm, rotated rx -180 ry 0 rz -180 deg; joints [-152.179, -41.789, -101.057, 33.508, 57.713, -19.477]
  Call Extruder(34168.21841)
  MoveL 3627 to (-49.52, 23.85, 155) mm, rotated rx 180 ry 0 rz 180 deg; joints [-153.248, -41.043, -102.867, 31.956, 58.264, -18.166]
  Call Extruder(34179.14855)
  MoveL 3628 to (-53.59, 12.23, 155) mm, rotated rx 180 ry 0 rz 180 deg; joints [-154.769, -40.442, -104.346, 29.974, 58.56, -16.743]
  Call Extruder(34190.07877)
  MoveL 3629 to (-54.97, 0, 155) mm, rotated rx -180 ry 0 rz -180 deg; joints [-156.673, -40.019, -105.4, 27.644, 58.589, -15.268]
  Call Extruder(34195.60439)
  MoveL 3630 to (-54.27, -6.18, 155) mm, rotated rx 180 ry 0 rz 180 deg; joints [-157.76, -39.902, -105.693, 26.363, 58.466, -14.531]
  Set speed (130.0 mm/s)
  MoveL 3631 to (-49.9, -9.51, 155) mm, rotated rx 180 ry 0 rz 180 deg; joints [-158.616, -40.091, -105.221, 25.464, 57.999, -14.163]
  MoveL 3632 to (-13.82, -4.92, 155) mm, rotated rx 180 ry 0 rz 180 deg; joints [-160.062, -42.572, -99.186, 24.79, 54.417, -15.043]
  Call Extruder(34228.77941)
  Set speed (20.0 mm/s)
  MoveL 3633 to (-4.92, -13.82, 155) mm, rotated rx 180 ry 0 rz -180 deg; joints [-161.89, -42.979, -98.224, 22.764, 53.45, -14.03]
  Call Extruder(34298.58601)
  MoveL 3634 to (13.82, 4.91, 155) mm, rotated rx -180 ry 0 rz -180 deg; joints [-160.09, -44.799, -93.997, 25.707, 51.73, -16.603]
  Call Extruder(34331.76103)
  MoveL 3635 to (4.92, 13.82, 155) mm, rotated rx -180 ry 0 rz -180 deg; joints [-158.352, -44.396, -94.924, 27.625, 52.709, -17.593]
  Set speed (130.0 mm/s)
  MoveL 3636 to (4.92, 13.82, 160) mm, rotated rx 180 ry 0 rz -180 deg; joints [-158.352, -43.672, -95.128, 27.811, 52.248, -17.898]
  Call Extruder(34329.76103)
  Set speed (40.0 mm/s)
  MoveL 3637 to (4.92, 13.82, 160) mm, rotated rx 180 ry 0 rz -180 deg; joints [-158.352, -43.672, -95.128, 27.811, 52.248, -17.898]
  Call Extruder(0.00000)
  Set speed (130.0 mm/s)
  MoveL 3638 to (-26.25, -4.54, 160) mm, rotated rx -180 ry 0 rz 180 deg; joints [-159.288, -40.96, -101.39, 25.527, 55.155, -15.262]
  Call Extruder(2.00000)
  Set speed (40.0 mm/s)
  MoveL 3639 to (-26.25, -4.54, 160) mm, rotated rx -180 ry 0 rz 180 deg; joints [-159.288, -40.96, -101.39, 25.527, 55.155, -15.262]
  Call Extruder(4.23262)
  Set speed (60.0 mm/s)
  MoveL 3640 to (-26.09, -5.96, 160) mm, rotated rx 180 ry 0 rz 180 deg; joints [-159.522, -40.935, -101.45, 25.242, 55.125, -15.087]
  Call Extruder(13.59741)
  MoveL 3641 to (-24.12, -11.61, 160) mm, rotated rx -180 ry 0 rz 180 deg; joints [-160.532, -40.929, -101.462, 24.048, 54.874, -14.399]
  Call Extruder(22.96233)
  MoveL 3642 to (-20.93, -16.69, 160) mm, rotated rx 180 ry 0 rz -180 deg; joints [-161.513, -41.029, -101.227, 22.919, 54.511, -13.791]
  Call Extruder(32.32753)
  MoveL 3643 to (-16.69, -20.93, 160) mm, rotated rx 180 ry 0 rz -180 deg; joints [-162.406, -41.228, -100.759, 21.923, 54.053, -13.293]
  Call Extruder(41.69245)
  MoveL 3644 to (-11.61, -24.12, 160) mm, rotated rx -180 ry 0 rz 180 deg; joints [-163.159, -41.516, -100.084, 21.118, 53.522, -12.932]
  Call Extruder(51.05724)
  MoveL 3645 to (-5.96, -26.09, 160) mm, rotated rx 180 ry 0 rz 180 deg; joints [-163.733, -41.879, -99.239, 20.548, 52.945, -12.728]
  Call Extruder(60.42235)
  MoveL 3646 to (0, -26.77, 160) mm, rotated rx 180 ry 0 rz 180 deg; joints [-164.103, -42.297, -98.271, 20.24, 52.348, -12.694]
  Call Extruder(69.78745)
  MoveL 3647 to (5.96, -26.09, 160) mm, rotated rx 180 ry 0 rz 180 deg; joints [-164.258, -42.749, -97.23, 20.207, 51.761, -12.834]
  Call Extruder(79.15226)
  MoveL 3648 to (11.61, -24.11, 160) mm, rotated rx 180 ry 0 rz 180 deg; joints [-164.201, -43.213, -96.17, 20.444, 51.215, -13.143]
  Call Extruder(88.51717)
  MoveL 3649 to (16.69, -20.93, 160) mm, rotated rx -180 ry 0 rz 180 deg; joints [-163.944, -43.665, -95.143, 20.93, 50.736, -13.607]
  Call Extruder(97.88238)
  MoveL 3650 to (20.93, -16.69, 160) mm, rotated rx 180 ry 0 rz 180 deg; joints [-163.508, -44.083, -94.199, 21.636, 50.35, -14.203]
  Call Extruder(107.24730)
  MoveL 3651 to (24.11, -11.61, 160) mm, rotated rx 180 ry 0 rz 180 deg; joints [-162.92, -44.446, -93.382, 22.519, 50.077, -14.899]
  Call Extruder(116.61209)
  MoveL 3652 to (26.09, -5.96, 160) mm, rotated rx 180 ry 0 rz -180 deg; joints [-162.209, -44.736, -92.731, 23.531, 49.932, -15.658]
  Call Extruder(125.97719)
  MoveL 3653 to (26.77, 0, 160) mm, rotated rx -180 ry 0 rz -180 deg; joints [-161.41, -44.94, -92.275, 24.621, 49.923, -16.439]
  Call Extruder(135.34229)
  MoveL 3654 to (26.09, 5.96, 160) mm, rotated rx 180 ry 0 rz 180 deg; joints [-160.556, -45.047, -92.036, 25.736, 50.051, -17.198]
  Call Extruder(144.70710)
  MoveL 3655 to (24.12, 11.61, 160) mm, rotated rx 180 ry 0 rz 180 deg; joints [-159.683, -45.052, -92.025, 26.822, 50.309, -17.896]
  Call Extruder(154.07201)
  MoveL 3656 to (20.93, 16.69, 160) mm, rotated rx 180 ry 0 rz 180 deg; joints [-158.826, -44.955, -92.242, 27.832, 50.683, -18.496]
  Call Extruder(163.43722)
  MoveL 3657 to (16.69, 20.93, 160) mm, rotated rx -180 ry 0 rz 180 deg; joints [-158.019, -44.76, -92.676, 28.724, 51.153, -18.97]
  Call Extruder(172.80213)
  MoveL 3658 to (11.61, 24.12, 160) mm, rotated rx 180 ry 0 rz 180 deg; joints [-157.299, -44.478, -93.309, 29.458, 51.696, -19.295]
  Call Extruder(182.16693)
  MoveL 3659 to (5.96, 26.09, 160) mm, rotated rx -180 ry 0 rz 180 deg; joints [-156.697, -44.121, -94.111, 30.006, 52.282, -19.458]
  Call Extruder(191.53204)
  MoveL 3660 to (0, 26.77, 160) mm, rotated rx 180 ry 0 rz 180 deg; joints [-156.245, -43.708, -95.045, 30.343, 52.883, -19.455]
  Call Extruder(200.89714)
  MoveL 3661 to (-5.96, 26.09, 160) mm, rotated rx 180 ry 0 rz 180 deg; joints [-155.969, -43.259, -96.066, 30.451, 53.467, -19.288]
  Call Extruder(210.26194)
  MoveL 3662 to (-11.61, 24.12, 160) mm, rotated rx -180 ry 0 rz -180 deg; joints [-155.891, -42.795, -97.125, 30.322, 54.007, -18.969]
  Call Extruder(219.62685)
  MoveL 3663 to (-16.69, 20.93, 160) mm, rotated rx 180 ry 0 rz -180 deg; joints [-156.025, -42.341, -98.17, 29.952, 54.475, -18.512]
  Call Extruder(228.99206)
  MoveL 3664 to (-20.93, 16.69, 160) mm, rotated rx 180 ry 0 rz 180 deg; joints [-156.374, -41.918, -99.148, 29.351, 54.848, -17.941]
  Call Extruder(238.35697)
  MoveL 3665 to (-24.11, 11.61, 160) mm, rotated rx -180 ry 0 rz 180 deg; joints [-156.928, -41.549, -100.007, 28.54, 55.109, -17.281]
  Call Extruder(247.72177)
  MoveL 3666 to (-26.09, 5.96, 160) mm, rotated rx -180 ry 0 rz 180 deg; joints [-157.665, -41.253, -100.701, 27.551, 55.245, -16.563]
  Call Extruder(257.08688)
  MoveL 3667 to (-26.77, 0, 160) mm, rotated rx 180 ry 0 rz 180 deg; joints [-158.546, -41.044, -101.191, 26.432, 55.251, -15.82]
  Call Extruder(261.87562)
  MoveL 3668 to (-26.42, -3.05, 160) mm, rotated rx 180 ry 0 rz 180 deg; joints [-159.044, -40.987, -101.326, 25.825, 55.186, -15.445]
  Call Extruder(259.87562)
  Set speed (40.0 mm/s)
  MoveL 3669 to (-26.42, -3.05, 160) mm, rotated rx 180 ry 0 rz 180 deg; joints [-159.044, -40.987, -101.326, 25.825, 55.186, -15.445]
  Call Extruder(0.00000)
  Set speed (130.0 mm/s)
  MoveL 3670 to (-41.86, -6.3, 160) mm, rotated rx 180 ry 0 rz 180 deg; joints [-158.606, -39.872, -103.982, 25.881, 56.688, -14.92]
  Call Extruder(2.00000)
  Set speed (40.0 mm/s)
  MoveL 3671 to (-41.86, -6.3, 160) mm, rotated rx 180 ry 0 rz 180 deg; joints [-158.606, -39.872, -103.982, 25.881, 56.688, -14.92]
  Call Extruder(6.99784)
  Set speed (60.0 mm/s)
  MoveL 3672 to (-41.5, -9.47, 160) mm, rotated rx 180 ry 0 rz 180 deg; joints [-159.151, -39.815, -104.119, 25.227, 56.622, -14.531]
  Call Extruder(21.89349)
  MoveL 3673 to (-38.36, -18.47, 160) mm, rotated rx 180 ry 0 rz 180 deg; joints [-160.835, -39.806, -104.14, 23.262, 56.225, -13.441]
  Call Extruder(36.78935)
  MoveL 3674 to (-33.28, -26.54, 160) mm, rotated rx -180 ry 0 rz 180 deg; joints [-162.466, -39.966, -103.755, 21.402, 55.652, -12.47]
  Call Extruder(51.68516)
  MoveL 3675 to (-26.54, -33.28, 160) mm, rotated rx -180 ry 0 rz -180 deg; joints [-163.93, -40.286, -102.99, 19.769, 54.928, -11.668]
  Call Extruder(66.58102)
  MoveL 3676 to (-18.47, -38.36, 160) mm, rotated rx -180 ry 0 rz 180 deg; joints [-165.137, -40.747, -101.892, 18.464, 54.089, -11.081]
  Call Extruder(81.47666)
  MoveL 3677 to (-9.47, -41.5, 160) mm, rotated rx -180 ry 0 rz 180 deg; joints [-166.024, -41.327, -100.527, 17.561, 53.174, -10.74]
  Call Extruder(96.37254)
  MoveL 3678 to (0, -42.57, 160) mm, rotated rx 180 ry 0 rz -180 deg; joints [-166.562, -41.994, -98.972, 17.098, 52.227, -10.671]
  Call Extruder(111.26841)
  MoveL 3679 to (9.47, -41.51, 160) mm, rotated rx -180 ry 0 rz 180 deg; joints [-166.745, -42.714, -97.31, 17.087, 51.293, -10.881]
  Call Extruder(126.16408)
  MoveL 3680 to (18.47, -38.36, 160) mm, rotated rx 180 ry 0 rz 180 deg; joints [-166.591, -43.452, -95.627, 17.51, 50.419, -11.366]
  Call Extruder(141.05992)
  MoveL 3681 to (26.54, -33.29, 160) mm, rotated rx -180 ry 0 rz 180 deg; joints [-166.133, -44.169, -94.004, 18.33, 49.651, -12.106]
  Call Extruder(155.95574)
  MoveL 3682 to (33.29, -26.54, 160) mm, rotated rx 180 ry 0 rz 180 deg; joints [-165.409, -44.831, -92.518, 19.49, 49.029, -13.065]
  Call Extruder(170.85159)
  MoveL 3683 to (38.36, -18.47, 160) mm, rotated rx -180 ry 0 rz 180 deg; joints [-164.468, -45.406, -91.236, 20.92, 48.588, -14.19]
  Call Extruder(185.74724)
  MoveL 3684 to (41.51, -9.47, 160) mm, rotated rx 180 ry 0 rz 180 deg; joints [-163.355, -45.866, -90.217, 22.54, 48.352, -15.42]
  Call Extruder(200.64312)
  MoveL 3685 to (42.57, 0, 160) mm, rotated rx 180 ry 0 rz 180 deg; joints [-162.12, -46.188, -89.504, 24.267, 48.336, -16.683]
  Call Extruder(215.53899)
  MoveL 3686 to (41.5, 9.47, 160) mm, rotated rx -180 ry 0 rz 180 deg; joints [-160.81, -46.358, -89.131, 26.015, 48.54, -17.907]
  Call Extruder(230.43465)
  MoveL 3687 to (38.36, 18.47, 160) mm, rotated rx 180 ry 0 rz 180 deg; joints [-159.475, -46.366, -89.113, 27.704, 48.955, -19.024]
  Call Extruder(245.33050)
  MoveL 3688 to (33.28, 26.54, 160) mm, rotated rx 180 ry 0 rz 180 deg; joints [-158.16, -46.212, -89.452, 29.263, 49.556, -19.975]
  Call Extruder(260.22632)
  MoveL 3689 to (26.54, 33.28, 160) mm, rotated rx 180 ry 0 rz 180 deg; joints [-156.916, -45.904, -90.132, 30.632, 50.311, -20.714]
  Call Extruder(275.12216)
  MoveL 3690 to (18.47, 38.36, 160) mm, rotated rx 180 ry 0 rz -180 deg; joints [-155.789, -45.457, -91.123, 31.76, 51.179, -21.21]
  Call Extruder(290.01783)
  MoveL 3691 to (9.47, 41.51, 160) mm, rotated rx 180 ry 0 rz -180 deg; joints [-154.828, -44.892, -92.381, 32.609, 52.116, -21.448]
  Call Extruder(304.91370)
  MoveL 3692 to (0, 42.57, 160) mm, rotated rx -180 ry 0 rz -180 deg; joints [-154.081, -44.237, -93.85, 33.147, 53.072, -21.423]
  Call Extruder(319.80957)
  MoveL 3693 to (-9.47, 41.51, 160) mm, rotated rx 180 ry 0 rz 180 deg; joints [-153.594, -43.524, -95.462, 33.347, 54.001, -21.145]
  Call Extruder(334.70523)
  MoveL 3694 to (-18.47, 38.36, 160) mm, rotated rx 180 ry 0 rz 180 deg; joints [-153.408, -42.787, -97.143, 33.19, 54.857, -20.633]
  Call Extruder(349.60108)
  MoveL 3695 to (-26.54, 33.29, 160) mm, rotated rx 180 ry 0 rz 180 deg; joints [-153.557, -42.064, -98.81, 32.664, 55.597, -19.912]
  Call Extruder(364.49689)
  MoveL 3696 to (-33.28, 26.54, 160) mm, rotated rx -180 ry 0 rz 180 deg; joints [-154.059, -41.39, -100.38, 31.769, 56.187, -19.014]
  Call Extruder(379.39274)
  MoveL 3697 to (-38.36, 18.47, 160) mm, rotated rx 180 ry 0 rz 180 deg; joints [-154.913, -40.8, -101.767, 30.522, 56.599, -17.981]
  Call Extruder(394.28840)
  MoveL 3698 to (-41.5, 9.47, 160) mm, rotated rx -180 ry 0 rz 180 deg; joints [-156.091, -40.326, -102.895, 28.965, 56.814, -16.855]
  Call Extruder(409.18428)
  MoveL 3699 to (-42.57, 0, 160) mm, rotated rx -180 ry 0 rz -180 deg; joints [-157.533, -39.991, -103.696, 27.168, 56.821, -15.688]
  Call Extruder(416.73856)
  MoveL 3700 to (-42.03, -4.8, 160) mm, rotated rx 180 ry 0 rz 180 deg; joints [-158.35, -39.899, -103.916, 26.187, 56.719, -15.102]
  Call Extruder(414.73856)
  Set speed (40.0 mm/s)
  MoveL 3701 to (-42.03, -4.8, 160) mm, rotated rx 180 ry 0 rz 180 deg; joints [-158.35, -39.899, -103.916, 26.187, 56.719, -15.102]
  Call Extruder(0.00000)
  Set speed (130.0 mm/s)
  MoveL 3702 to (-54.1, -7.67, 160) mm, rotated rx 180 ry 0 rz -180 deg; joints [-158.024, -39.049, -105.981, 26.218, 57.893, -14.668]
  Call Extruder(2.00000)
  Set speed (40.0 mm/s)
  MoveL 3703 to (-54.1, -7.67, 160) mm, rotated rx 180 ry 0 rz -180 deg; joints [-158.024, -39.049, -105.981, 26.218, 57.893, -14.668]
  Call Extruder(6.07263)
  Set speed (30.0 mm/s)
  MoveL 3704 to (-53.59, -12.23, 160) mm, rotated rx 180 ry 0 rz 180 deg; joints [-158.835, -38.967, -106.181, 25.258, 57.798, -14.113]
  Call Extruder(17.00276)
  MoveL 3705 to (-49.53, -23.85, 160) mm, rotated rx 180 ry 0 rz 180 deg; joints [-161.095, -38.956, -106.208, 22.648, 57.289, -12.707]
  Call Extruder(27.93305)
  MoveL 3706 to (-42.98, -34.27, 160) mm, rotated rx 180 ry 0 rz 180 deg; joints [-163.275, -39.164, -105.699, 20.176, 56.552, -11.449]
  Call Extruder(38.86316)
  MoveL 3707 to (-34.27, -42.98, 160) mm, rotated rx 180 ry 0 rz 180 deg; joints [-165.21, -39.579, -104.688, 18.017, 55.622, -10.406]
  Call Extruder(49.79345)
  MoveL 3708 to (-23.85, -49.53, 160) mm, rotated rx 180 ry 0 rz 180 deg; joints [-166.774, -40.179, -103.245, 16.313, 54.544, -9.635]
  Call Extruder(60.72358)
  MoveL 3709 to (-12.23, -53.59, 160) mm, rotated rx -180 ry 0 rz 180 deg; joints [-167.889, -40.93, -101.46, 15.157, 53.366, -9.181]
  Call Extruder(71.65380)
  MoveL 3710 to (0, -54.97, 160) mm, rotated rx -180 ry 0 rz 180 deg; joints [-168.526, -41.793, -99.438, 14.592, 52.145, -9.077]
  Call Extruder(82.58402)
  MoveL 3711 to (12.23, -53.59, 160) mm, rotated rx 180 ry 0 rz 180 deg; joints [-168.697, -42.724, -97.288, 14.621, 50.938, -9.336]
  Call Extruder(93.51417)
  MoveL 3712 to (23.85, -49.53, 160) mm, rotated rx -180 ry 0 rz 180 deg; joints [-168.436, -43.675, -95.12, 15.214, 49.806, -9.955]
  Call Extruder(104.44444)
  MoveL 3713 to (34.27, -42.98, 160) mm, rotated rx 180 ry 0 rz 180 deg; joints [-167.797, -44.599, -93.037, 16.314, 48.806, -10.911]
  Call Extruder(115.37457)
  MoveL 3714 to (42.98, -34.27, 160) mm, rotated rx -180 ry 0 rz 180 deg; joints [-166.837, -45.452, -91.133, 17.846, 47.994, -12.158]
  Call Extruder(126.30485)
